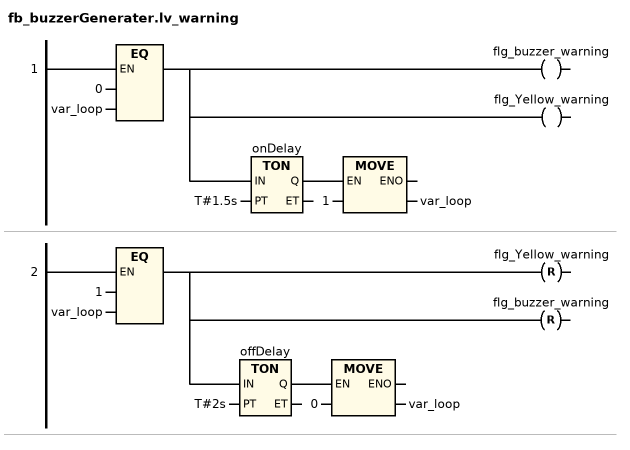
// NETWORK 1
_w3 := 0 = var_loop;
flg_buzzer_warning := _w3;
flg_Yellow_warning := _w3;
onDelay(IN := _w3, PT := T#1.5s); // TON
IF onDelay.Q THEN var_loop := 1; END_IF

// NETWORK 2
_w4 := 1 = var_loop;
flg_Yellow_warning R= _w4;
flg_buzzer_warning R= _w4;
offDelay(IN := _w4, PT := T#2s); // TON
IF offDelay.Q THEN var_loop := 0; END_IF
END_ACTION

ACTION manual:
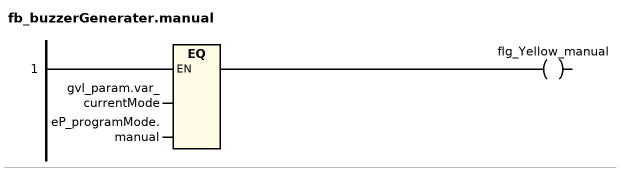
// NETWORK 1
flg_Yellow_manual := gvl_param.var_currentMode = eP_programMode.manual;
END_ACTION

END_FUNCTION_BLOCK

// ---- FBs/fb_eleControllers.TcPOU
FUNCTION_BLOCK fb_eleControllers
VAR_INPUT
END_VAR
VAR_OUTPUT
END_VAR
VAR
END_VAR

gvl_elecylinder.fbi_axisTransport(
	var_ref_ele:= gvl_elecylinder.ref_axis_transport, 
	in_flg_run:= , 
	in_var_moveMode:= , 
	in_flg_pause:= , 
	out_flg_run=> , 
	out_flg_busy=> , 
	out_flg_Done=> , 
	out_flg_error=> );
gvl_elecylinder.fbi_axisSample(
	var_ref_ele:= gvl_elecylinder.ref_axis_sample, 
	in_flg_run:= , 
	in_var_moveMode:= , 
	in_flg_pause:= NOT gvl_io.flg_frontSaftyDoor AND gvl_param.var_currentMode = eP_programMode.auto, 
	out_flg_run=> , 
	out_flg_busy=> , 
	out_flg_Done=> , 
	out_flg_error=> );
gvl_elecylinder.fbi_axisTrayChange(
	var_ref_ele:= gvl_elecylinder.ref_axis_trayChange, 
	in_flg_run:= , 
	in_var_moveMode:= , 
	in_flg_pause:=  NOT gvl_io.flg_frontSaftyDoor AND gvl_param.var_currentMode = eP_programMode.auto, 
	out_flg_run=> , 
	out_flg_busy=> , 
	out_flg_Done=> , 
	out_flg_error=> );
gvl_elecylinder.fbi_axisRotary(
	var_ref_ele:= gvl_elecylinder.ref_axis_rotary, 
	in_flg_run:= , 
	in_var_moveMode:= , 
	in_flg_pause:= , 
	out_flg_run=> , 
	out_flg_busy=> , 
	out_flg_Done=> , 
	out_flg_error=> );
gvl_elecylinder.fbi_gm_axisPickUp(
	var_ref_ele:= gvl_elecylinder.ref_gm_axisPickUp, 
	in_flg_run:= , 
	in_var_moveMode:= , 
	in_flg_pause:= , 
	out_flg_run=> , 
	out_flg_busy=> , 
	out_flg_Done=> , 
	out_flg_error=> );
gvl_elecylinder.fbi_gm_axisTransport(
	var_ref_ele:= gvl_elecylinder.ref_gm_axisTransport, 
	in_flg_run:= , 
	in_var_moveMode:= , 
	in_flg_pause:= , 
	out_flg_run=> , 
	out_flg_busy=> , 
	out_flg_Done=> , 
	out_flg_error=> );
	
IF gvl_elecylinder.ref_axis_trayChange.input.in_flg_sensA THEN
	gvl_param.var_currentTrayPos := 1;
	gvl_visu.var_currentTableMsg := "上段";
ELSIF gvl_elecylinder.ref_axis_trayChange.input.in_flg_sensB THEN
	gvl_param.var_currentTrayPos := 2;
	gvl_visu.var_currentTableMsg := "下段";
ELSE 
	gvl_param.var_currentTrayPos := 0;
	gvl_visu.var_currentTableMsg := "テーブル移動中...";
END_IF

END_FUNCTION_BLOCK

// ---- FBs/fb_svControllers.TcPOU
FUNCTION_BLOCK fb_svControllers
VAR_INPUT
END_VAR
VAR_OUTPUT
END_VAR
VAR
END_VAR

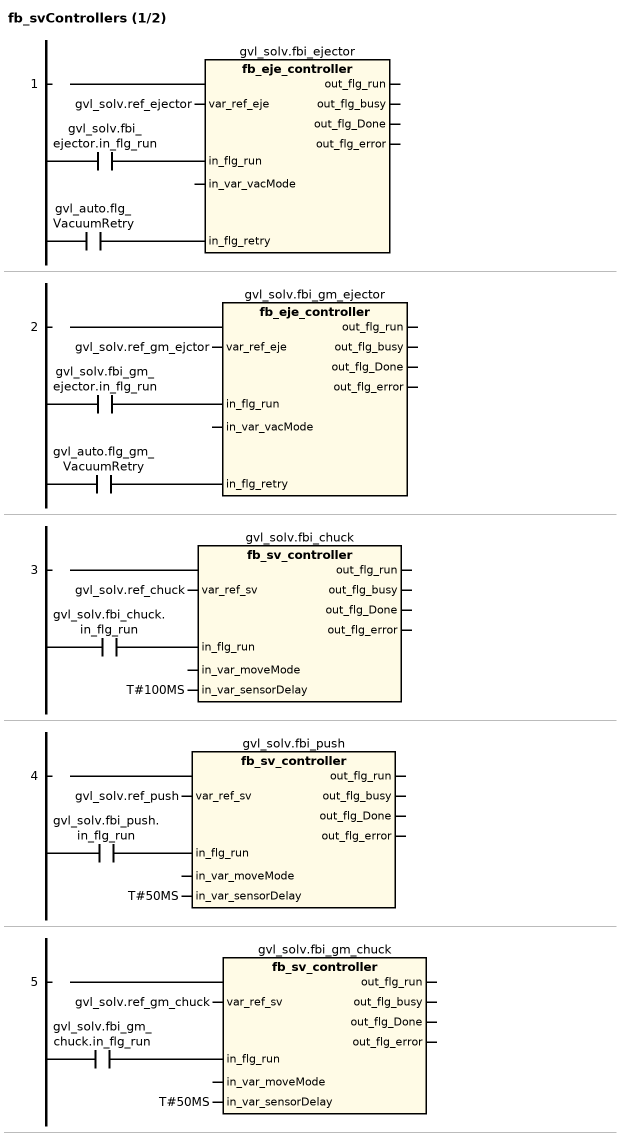
// NETWORK 1
gvl_solv.fbi_ejector(
    var_ref_eje := gvl_solv.ref_ejector,
    in_flg_run := gvl_solv.fbi_ejector.in_flg_run,
    in_flg_retry := gvl_auto.flg_VacuumRetry); // fb_eje_controller

// NETWORK 2
gvl_solv.fbi_gm_ejector(
    var_ref_eje := gvl_solv.ref_gm_ejctor,
    in_flg_run := gvl_solv.fbi_gm_ejector.in_flg_run,
    in_flg_retry := gvl_auto.flg_gm_VacuumRetry); // fb_eje_controller

// NETWORK 3
gvl_solv.fbi_chuck(
    var_ref_sv := gvl_solv.ref_chuck,
    in_flg_run := gvl_solv.fbi_chuck.in_flg_run,
    in_var_sensorDelay := T#100MS); // fb_sv_controller

// NETWORK 4
gvl_solv.fbi_push(
    var_ref_sv := gvl_solv.ref_push,
    in_flg_run := gvl_solv.fbi_push.in_flg_run,
    in_var_sensorDelay := T#50MS); // fb_sv_controller

// NETWORK 5
gvl_solv.fbi_gm_chuck(
    var_ref_sv := gvl_solv.ref_gm_chuck,
    in_flg_run := gvl_solv.fbi_gm_chuck.in_flg_run,
    in_var_sensorDelay := T#50MS); // fb_sv_controller

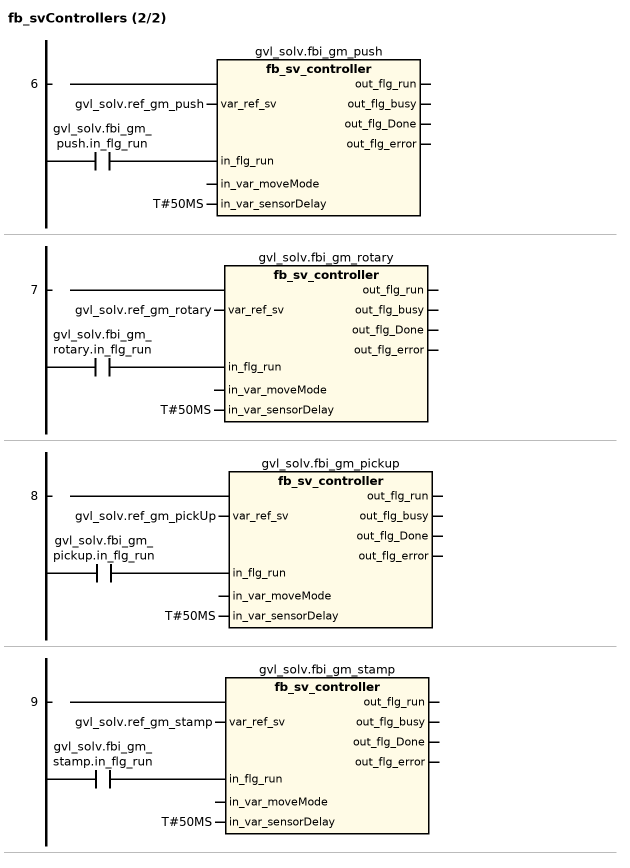
// NETWORK 6
gvl_solv.fbi_gm_push(
    var_ref_sv := gvl_solv.ref_gm_push,
    in_flg_run := gvl_solv.fbi_gm_push.in_flg_run,
    in_var_sensorDelay := T#50MS); // fb_sv_controller

// NETWORK 7
gvl_solv.fbi_gm_rotary(
    var_ref_sv := gvl_solv.ref_gm_rotary,
    in_flg_run := gvl_solv.fbi_gm_rotary.in_flg_run,
    in_var_sensorDelay := T#50MS); // fb_sv_controller

// NETWORK 8
gvl_solv.fbi_gm_pickup(
    var_ref_sv := gvl_solv.ref_gm_pickUp,
    in_flg_run := gvl_solv.fbi_gm_pickup.in_flg_run,
    in_var_sensorDelay := T#50MS); // fb_sv_controller

// NETWORK 9
gvl_solv.fbi_gm_stamp(
    var_ref_sv := gvl_solv.ref_gm_stamp,
    in_flg_run := gvl_solv.fbi_gm_stamp.in_flg_run,
    in_var_sensorDelay := T#50MS); // fb_sv_controller

END_FUNCTION_BLOCK

// ---- FBs/fb_ejecter/fb_eje_controller.TcPOU
FUNCTION_BLOCK fb_eje_controller
VAR_IN_OUT
	var_ref_eje : ref_eje_io;
END_VAR
VAR_INPUT
	in_flg_run : BOOL;
	in_var_vacMode : eP_ejeVacMode;
	in_flg_retry: BOOL;
END_VAR
VAR_OUTPUT
	out_flg_run : BOOL;
	out_flg_busy: BOOL;
	out_flg_Done: BOOL;
	out_flg_error : BOOL;
END_VAR
VAR
	var_buf_moveMode: eP_ejeVacMode;
	flg_vacOnDone: BOOL;
	flg_vacOffDone: BOOL;
	flg_vacBreakDone: BOOL;
	flg_vacHaltDone: BOOL;
	fbi_brakTime: TON;
	flg_breakDone: BOOL;
	var_timeOut: TON;
	in: BOOL;
END_VAR
VAR // added by the converter: edge detectors and wires of the graphical bodies
    _rt1, _rt2, _rt3, _rt4 : R_TRIG;
    _w1, _w2, _w3, _w4, _w5 : BOOL;
END_VAR

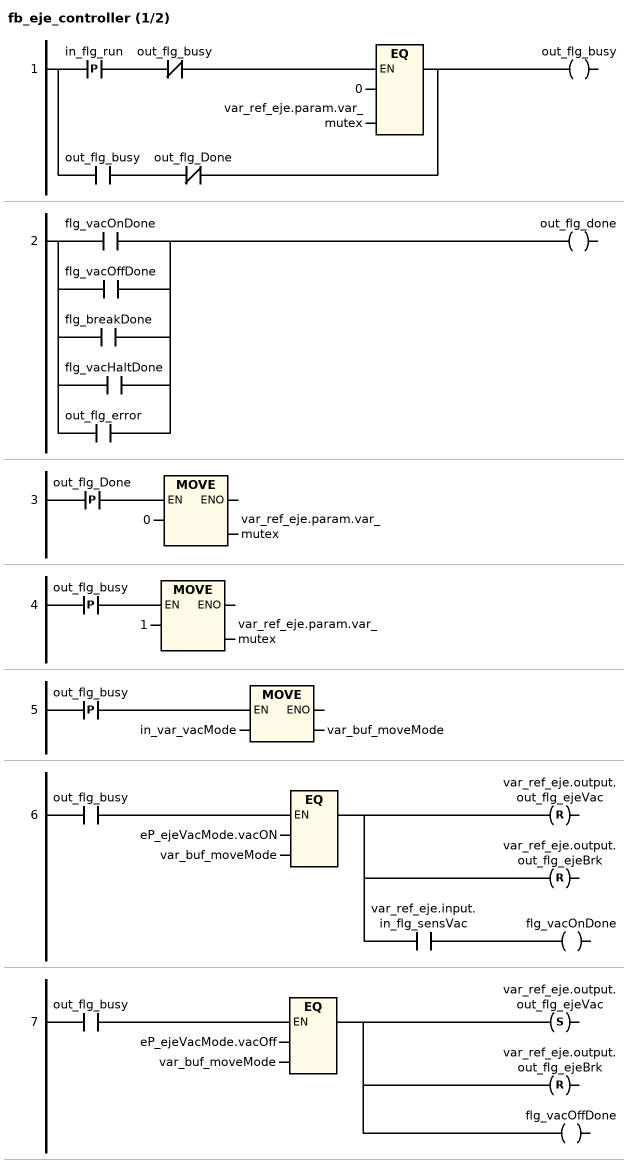
// NETWORK 1
_rt1(CLK := in_flg_run);
out_flg_busy := _rt1.Q AND NOT out_flg_busy AND 0 = var_ref_eje.param.var_mutex OR out_flg_busy AND NOT out_flg_Done;

// NETWORK 2
out_flg_done := flg_vacOnDone OR flg_vacOffDone OR flg_breakDone OR flg_vacHaltDone OR out_flg_error;

// NETWORK 3
_rt2(CLK := out_flg_Done);
IF _rt2.Q THEN var_ref_eje.param.var_mutex := 0; END_IF

// NETWORK 4
_rt3(CLK := out_flg_busy);
IF _rt3.Q THEN var_ref_eje.param.var_mutex := 1; END_IF

// NETWORK 5
_rt4(CLK := out_flg_busy);
IF _rt4.Q THEN var_buf_moveMode := in_var_vacMode; END_IF

// NETWORK 6
_w1 := out_flg_busy AND eP_ejeVacMode.vacON = var_buf_moveMode;
var_ref_eje.output.out_flg_ejeVac R= _w1;
var_ref_eje.output.out_flg_ejeBrk R= _w1;
flg_vacOnDone := _w1 AND var_ref_eje.input.in_flg_sensVac;

// NETWORK 7
_w2 := out_flg_busy AND eP_ejeVacMode.vacOff = var_buf_moveMode;
var_ref_eje.output.out_flg_ejeVac S= _w2;
var_ref_eje.output.out_flg_ejeBrk R= _w2;
flg_vacOffDone := _w2;

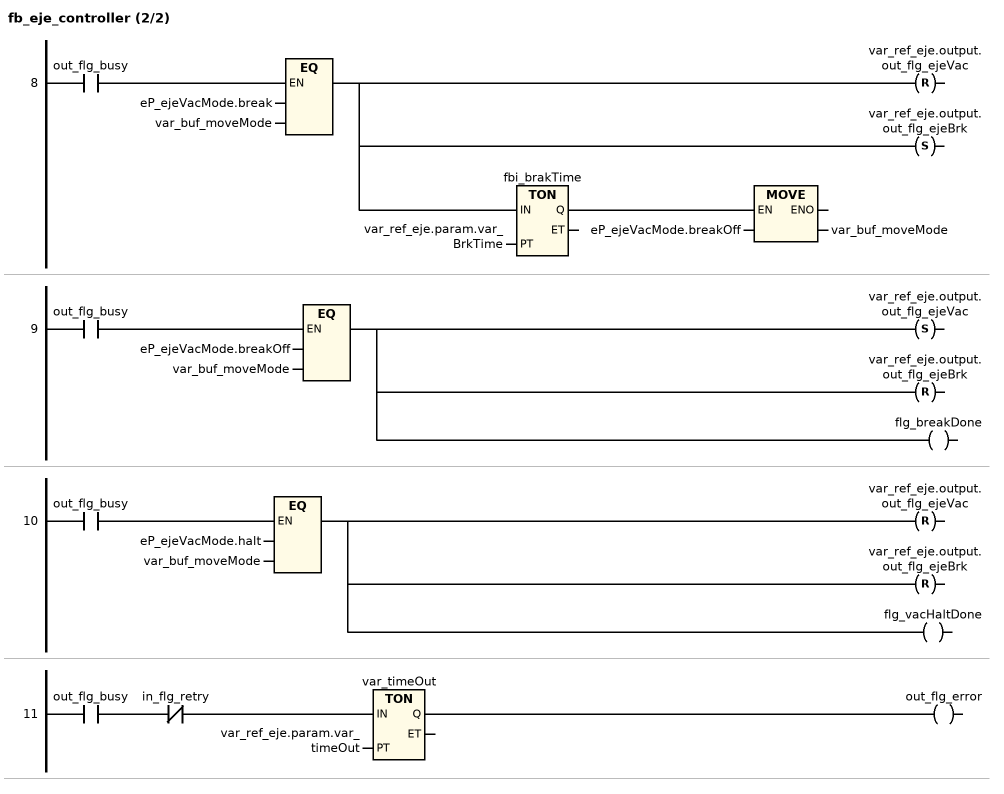
// NETWORK 8
_w3 := out_flg_busy AND eP_ejeVacMode.break = var_buf_moveMode;
var_ref_eje.output.out_flg_ejeVac R= _w3;
var_ref_eje.output.out_flg_ejeBrk S= _w3;
fbi_brakTime(IN := _w3, PT := var_ref_eje.param.var_BrkTime); // TON
IF fbi_brakTime.Q THEN var_buf_moveMode := eP_ejeVacMode.breakOff; END_IF

// NETWORK 9
_w4 := out_flg_busy AND eP_ejeVacMode.breakOff = var_buf_moveMode;
var_ref_eje.output.out_flg_ejeVac S= _w4;
var_ref_eje.output.out_flg_ejeBrk R= _w4;
flg_breakDone := _w4;

// NETWORK 10
_w5 := out_flg_busy AND eP_ejeVacMode.halt = var_buf_moveMode;
var_ref_eje.output.out_flg_ejeVac R= _w5;
var_ref_eje.output.out_flg_ejeBrk R= _w5;
flg_vacHaltDone := _w5;

// NETWORK 11
var_timeOut(IN := out_flg_busy AND NOT in_flg_retry, PT := var_ref_eje.param.var_timeOut); // TON
out_flg_error := var_timeOut.Q;

END_FUNCTION_BLOCK

// ---- FBs/fb_sv/fb_sv_controller.TcPOU
FUNCTION_BLOCK fb_sv_controller
VAR_IN_OUT
	var_ref_sv : ref_sv_io;
END_VAR
VAR_INPUT
	in_flg_run : BOOL;
	in_var_moveMode : eP_svMoveMode;
	in_var_sensorDelay : TIME;
END_VAR
VAR_OUTPUT
	out_flg_run : BOOL;
	out_flg_busy: BOOL;
	out_flg_Done: BOOL;
	out_flg_error : BOOL;
END_VAR
VAR
	var_buf_moveMode: eP_svMoveMode;
	fbi_sensorDelayTimerA: TON;
	fbi_sensorDelayTimerB: TON;
	flg_svADone: BOOL;
	flg_svBDone: BOOL;
	fbi_timeOut: TON;
	flg_svSDone: BOOL;
END_VAR
VAR // added by the converter: edge detectors and wires of the graphical bodies
    _rt1, _rt2, _rt3, _rt4 : R_TRIG;
    _w1, _w2, _w3 : BOOL;
END_VAR

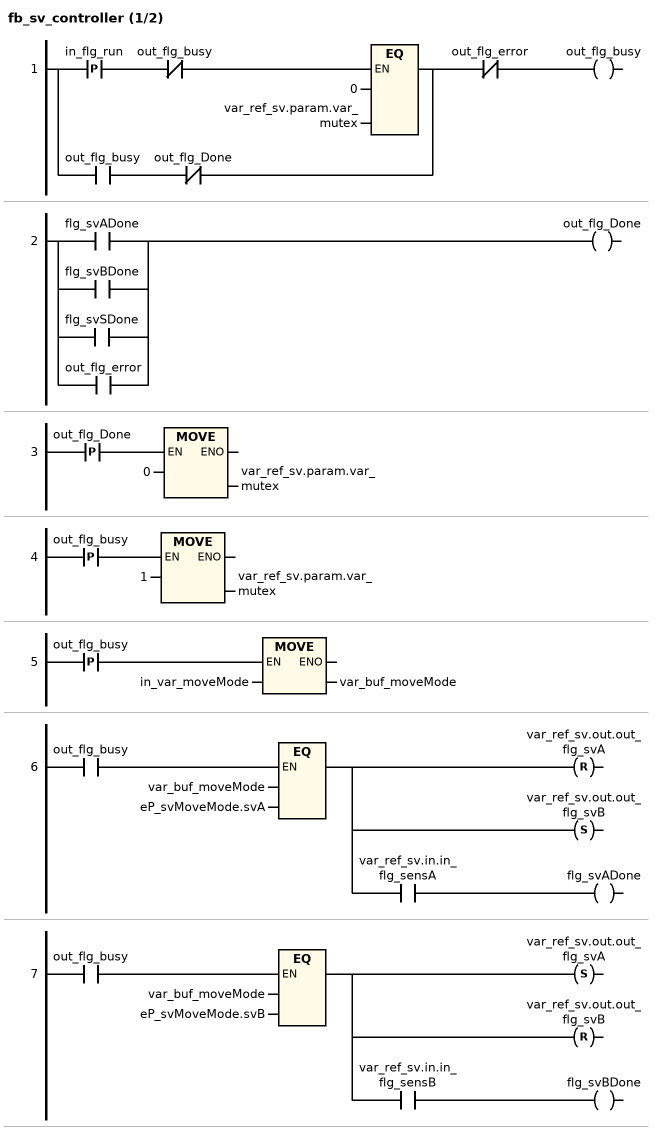
// NETWORK 1
_rt1(CLK := in_flg_run);
out_flg_busy := (_rt1.Q AND NOT out_flg_busy AND 0 = var_ref_sv.param.var_mutex OR out_flg_busy AND NOT out_flg_Done) AND NOT out_flg_error;

// NETWORK 2
out_flg_Done := flg_svADone OR flg_svBDone OR flg_svSDone OR out_flg_error;

// NETWORK 3
_rt2(CLK := out_flg_Done);
IF _rt2.Q THEN var_ref_sv.param.var_mutex := 0; END_IF

// NETWORK 4
_rt3(CLK := out_flg_busy);
IF _rt3.Q THEN var_ref_sv.param.var_mutex := 1; END_IF

// NETWORK 5
_rt4(CLK := out_flg_busy);
IF _rt4.Q THEN var_buf_moveMode := in_var_moveMode; END_IF

// NETWORK 6
_w1 := out_flg_busy AND var_buf_moveMode = eP_svMoveMode.svA;
var_ref_sv.out.out_flg_svA R= _w1;
var_ref_sv.out.out_flg_svB S= _w1;
flg_svADone := _w1 AND var_ref_sv.in.in_flg_sensA;

// NETWORK 7
_w2 := out_flg_busy AND var_buf_moveMode = eP_svMoveMode.svB;
var_ref_sv.out.out_flg_svA S= _w2;
var_ref_sv.out.out_flg_svB R= _w2;
flg_svBDone := _w2 AND var_ref_sv.in.in_flg_sensB;

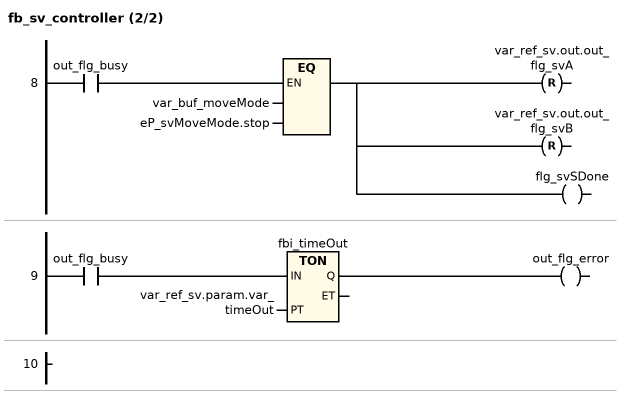
// NETWORK 8
_w3 := out_flg_busy AND var_buf_moveMode = eP_svMoveMode.stop;
var_ref_sv.out.out_flg_svA R= _w3;
var_ref_sv.out.out_flg_svB R= _w3;
flg_svSDone := _w3;

// NETWORK 9
fbi_timeOut(IN := out_flg_busy, PT := var_ref_sv.param.var_timeOut); // TON
out_flg_error := fbi_timeOut.Q;

// NETWORK 10

END_FUNCTION_BLOCK

// ---- FBs/fb_sampleSchedule.TcPOU
FUNCTION_BLOCK fb_sampleSchedule
VAR_INPUT
	in_var_enableSchedule: ARRAY[0..6] OF BOOL;
	in_var_scheduleTimeH : ARRAY[0..6] OF WORD;
	in_var_scheduleTimeM : ARRAY[0..6] OF WORD;
END_VAR
VAR_OUTPUT
	out_flg_sampletriger : bool;
END_VAR
VAR
	fbi_GetLocalAmsNetId : FB_GetLocalAmsNetId;
	fbi_LocalSystemTime : FB_LocalSystemTime;
	var_scheduleTime : ARRAY[0..6] OF s_timeSchedule;
	var_scheduleNumber : INT;
	fbi_r_trig: R_TRIG;
	var_process: INT;
END_VAR

fbi_GetLocalAmsNetId(
	bExecute:= TRUE, 
	tTimeOut:= , 
	bBusy=> , 
	bError=> , 
	nErrId=> , 
	AddrString=> , 
	AddrBytes=> );
fbi_LocalSystemTime(
	sNetID:=fbi_GetLocalAmsNetId.AddrString , 
	bEnable:= TRUE, 
	dwCycle:= , 
	dwOpt:= , 
	tTimeout:= , 
	bValid=> , 
	systemTime=> ,
	tzID=> );
fbi_r_trig(CLK:= , Q=> );
FOR var_scheduleNumber := 0 TO 6 BY 1 DO
	IF in_var_enableSchedule[var_scheduleNumber] THEN
		var_scheduleTime[var_scheduleNumber].hour := in_var_scheduleTimeH[var_scheduleNumber];
		var_scheduleTime[var_scheduleNumber].minute := in_var_scheduleTimeM[var_scheduleNumber];
		IF fbi_LocalSystemTime.systemTime.wHour = var_scheduleTime[var_scheduleNumber].hour THEN
			IF fbi_LocalSystemTime.systemTime.wMinute = var_scheduleTime[var_scheduleNumber].minute THEN		
				fbi_r_trig.CLK := TRUE;
			ELSE
				fbi_r_trig.CLK := FALSE;
			END_IF
		END_IF
	END_IF
END_FOR
out_flg_sampletriger := fbi_r_trig.Q;

END_FUNCTION_BLOCK

// ---- FBs/fb_text_control.TcPOU
FUNCTION_BLOCK fb_text_control
VAR_INPUT
END_VAR
VAR_OUTPUT
END_VAR
VAR
END_VAR

IF gvl_param.var_currentMode = eP_programMode.auto THEN
	IF gvl_debug.out_busy THEN
		gvl_text.var_auto_runing := "デバッグ運転中";
	ELSE
		gvl_text.var_auto_runing := "自動運転中";
	END_IF
ELSE
	gvl_text.var_auto_runing := "自動運転開始";
END_IF
IF gvl_auto.autoModeStop THEN
	gvl_text.var_stopping:= "自動運転停止中";
ELSE
	gvl_text.var_stopping:= "自動運転停止";
END_IF
IF gvl_visu.flg_btn_trayChangeDone THEN
	gvl_text.var_trayChangeDone:= "トレイ交換完了済";
ELSE
	gvl_text.var_trayChangeDone:= "トレイ交換完了";
END_IF

END_FUNCTION_BLOCK

// ---- FBs/fb_motionController.TcPOU
FUNCTION_BLOCK fb_motionController
VAR_INPUT
	in_flg_run : BOOL;
END_VAR
VAR_OUTPUT
	out_flg_run : BOOL;
END_VAR
VAR_IN_OUT
	var_ref_X : ref_mc_moveAbs;
	var_ref_Y : ref_mc_moveAbs;
	var_ref_Z : ref_mc_moveAbs;
END_VAR
VAR_INPUT
	in_flg_start : BOOL;
	in_var_targetPosX : LREAL;
	in_var_targetPosY : LREAL;
	in_var_targetPosZ : LREAL;
	in_var_direction : eP_motionDirection;
	
END_VAR
VAR_OUTPUT
	out_flg_busy : BOOL;
	out_flg_Done : BOOL;
	out_flg_moveXYDone : BOOL;
	
END_VAR
VAR
	SFCInit : BOOL;
	fbi_r_TIRG: R_TRIG;
	fbi_f_TRIG: F_TRIG;
	var_buf_targetPosX: LREAL;
	var_buf_targetPosY: LREAL;
	var_buf_targetPosZ: LREAL;
	var_buf_direction: eP_motionDirection;
	trn_getParamDone: BOOL;
	var_mutex: INT;
	trn_moveXY_1Done: BOOL;
	trn_moveZ_1Done: BOOL;
	trn_moveZ_2Done: BOOL;
	trn_moveXY_2Done: BOOL;
	
	trn_moveX_3Done: BOOL;
	trn_moveY_3Done: BOOL;
	trn_moveZ_3Done: BOOL;
	
	trn_moveX_4Done: BOOL;
	trn_moveY_4Done: BOOL;
	trn_moveZ_4Done: BOOL;

	trn_executeReset2Done: BOOL;
	var_process: INT;
END_VAR

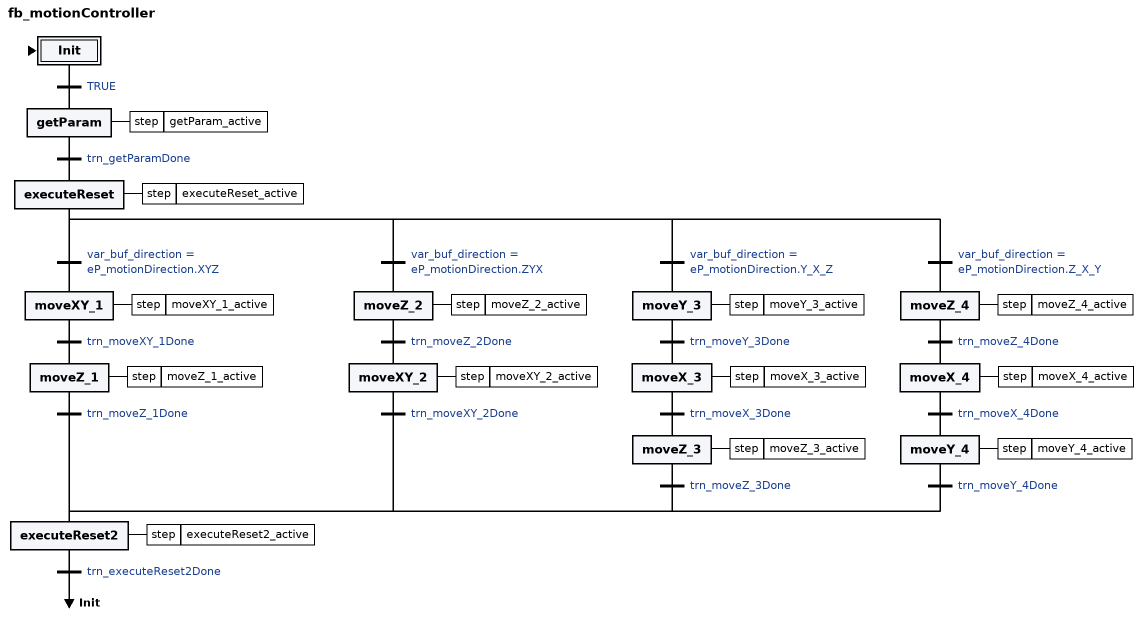
INITIAL_STEP Init:
END_STEP
TRANSITION FROM Init TO getParam
    := TRUE;
END_TRANSITION
STEP getParam:
    getParam_active(N);  // step action
END_STEP
TRANSITION FROM getParam TO executeReset
    := trn_getParamDone;
END_TRANSITION
STEP executeReset:
    executeReset_active(N);  // step action
END_STEP
TRANSITION FROM executeReset TO moveXY_1
    := var_buf_direction = eP_motionDirection.XYZ;
END_TRANSITION
STEP moveXY_1:
    moveXY_1_active(N);  // step action
END_STEP
TRANSITION FROM moveXY_1 TO moveZ_1
    := trn_moveXY_1Done;
END_TRANSITION
STEP moveZ_1:
    moveZ_1_active(N);  // step action
END_STEP
TRANSITION FROM moveZ_1 TO executeReset2
    := trn_moveZ_1Done;
END_TRANSITION
TRANSITION FROM executeReset TO moveZ_2
    := var_buf_direction = eP_motionDirection.ZYX;
END_TRANSITION
STEP moveZ_2:
    moveZ_2_active(N);  // step action
END_STEP
TRANSITION FROM moveZ_2 TO moveXY_2
    := trn_moveZ_2Done;
END_TRANSITION
STEP moveXY_2:
    moveXY_2_active(N);  // step action
END_STEP
TRANSITION FROM moveXY_2 TO executeReset2
    := trn_moveXY_2Done;
END_TRANSITION
TRANSITION FROM executeReset TO moveY_3
    := var_buf_direction = eP_motionDirection.Y_X_Z;
END_TRANSITION
STEP moveY_3:
    moveY_3_active(N);  // step action
END_STEP
TRANSITION FROM moveY_3 TO moveX_3
    := trn_moveY_3Done;
END_TRANSITION
STEP moveX_3:
    moveX_3_active(N);  // step action
END_STEP
TRANSITION FROM moveX_3 TO moveZ_3
    := trn_moveX_3Done;
END_TRANSITION
STEP moveZ_3:
    moveZ_3_active(N);  // step action
END_STEP
TRANSITION FROM moveZ_3 TO executeReset2
    := trn_moveZ_3Done;
END_TRANSITION
TRANSITION FROM executeReset TO moveZ_4
    := var_buf_direction = eP_motionDirection.Z_X_Y;
END_TRANSITION
STEP moveZ_4:
    moveZ_4_active(N);  // step action
END_STEP
TRANSITION FROM moveZ_4 TO moveX_4
    := trn_moveZ_4Done;
END_TRANSITION
STEP moveX_4:
    moveX_4_active(N);  // step action
END_STEP
TRANSITION FROM moveX_4 TO moveY_4
    := trn_moveX_4Done;
END_TRANSITION
STEP moveY_4:
    moveY_4_active(N);  // step action
END_STEP
TRANSITION FROM moveY_4 TO executeReset2
    := trn_moveY_4Done;
END_TRANSITION
STEP executeReset2:
    executeReset2_active(N);  // step action
END_STEP
TRANSITION FROM executeReset2 TO Init
    := trn_executeReset2Done;
END_TRANSITION

ACTION executeReset_active:
IF executeReset._x AND executeReset.x = FALSE THEN
	var_ref_x.Execute := FALSE;
	var_ref_y.Execute := FALSE;
	var_ref_z.Execute := FALSE;
ELSIF executeReset._x AND executeReset.x THEN
	var_ref_x.Execute := FALSE;
	var_ref_y.Execute := FALSE;
	var_ref_z.Execute := FALSE;
END_IF
END_ACTION

ACTION executeReset2_active:
IF executeReset2._x AND executeReset2.x= FALSE THEN
	trn_executeReset2Done := FALSE;
	var_ref_x.Execute := FALSE;
	var_ref_y.Execute := FALSE;
	var_ref_z.Execute := FALSE;
	out_flg_done := TRUE;
	out_flg_moveXYDone := FALSE;
ELSIF executeReset2._x AND executeReset2.x THEN
	var_ref_x.Execute := FALSE;
	var_ref_y.Execute := FALSE;
	var_ref_z.Execute := FALSE;
	trn_executeReset2Done := TRUE;
	out_flg_done := FALSE;
	in_flg_start := FALSE;
END_IF
END_ACTION

ACTION getParam_active:
fbi_r_TIRG(CLK:= in_flg_start, Q=> );
IF getParam._x AND getParam.x = FALSE THEN
	var_mutex := 0;
	trn_getParamDone := FALSE;
	out_flg_moveXYDone:= FALSE;
	in_flg_start := FALSE;
ELSIF getParam._x AND getParam.x THEN
	IF fbi_r_TIRG.Q THEN
		var_ref_x.Position := in_var_targetPosX;
		var_ref_Y.Position := in_var_targetPosY;
		var_ref_Z.Position := in_var_targetPosZ;
		var_buf_direction := in_var_direction;
		var_mutex := 1;
	END_IF
	IF var_mutex = 1 THEN
		out_flg_busy := TRUE;
		trn_getParamDone := TRUE;
	ELSE
		out_flg_busy := FALSE;
		trn_getParamDone := FALSE;
	END_IF
	IF in_flg_run THEN
		out_flg_run := TRUE;
	ELSE
		out_flg_run := FALSE;
	END_IF
END_IF
END_ACTION

ACTION moveX_3_active:
IF moveX_3._x AND moveX_3.x = FALSE THEN
	trn_moveX_3Done := FALSE;
	var_process := 0;
ELSIF moveX_3._x AND moveX_3.x THEN
	CASE var_process OF
		0:
			var_ref_x.Execute := TRUE;
			var_process := 1;
		1:
			IF var_ref_x.Done THEN
				trn_moveX_3Done := TRUE;
			END_IF
	END_CASE
END_IF
END_ACTION

ACTION moveX_4_active:
IF moveX_4._x AND moveX_4.x = FALSE THEN
	trn_moveX_4Done := FALSE;
	var_process := 0;
ELSIF moveX_4._x AND moveX_4.x THEN
	CASE var_process OF
		0:
			var_ref_x.Execute := TRUE;
			var_process := 1;
		1:
			IF var_ref_x.Done THEN
				trn_moveX_4Done := TRUE;
			END_IF
	END_CASE
END_IF
END_ACTION

ACTION moveXY_1_active:
IF moveXY_1._x AND moveXY_1.x = FALSE THEN
	out_flg_moveXYDone:= FALSE;
	trn_moveXY_1Done := FALSE;
	var_process := 0;
ELSIF moveXY_1._x AND moveXY_1.x THEN
	CASE var_process OF
		0:
			var_ref_x.Execute := TRUE;
			var_ref_y.Execute := TRUE;
			var_process := 1;
		1:
			IF var_ref_x.Done AND var_ref_y.Done THEN
				out_flg_moveXYDone:= TRUE;
				trn_moveXY_1Done := TRUE;
			END_IF
	END_CASE
END_IF
END_ACTION

ACTION moveXY_2_active:
IF moveXY_2._x AND moveXY_2.x = FALSE THEN
	trn_moveXY_2Done := FALSE;
	var_process := 0;
ELSIF moveXY_2._x AND moveXY_2.x THEN
	CASE var_process OF
		0:
			var_ref_x.Execute := TRUE;
			var_ref_y.Execute := TRUE;
			var_process := 1;
		1:
			IF var_ref_x.Done AND var_ref_y.Done THEN
				trn_moveXY_2Done := TRUE;
			END_IF
	END_CASE
END_IF
END_ACTION

ACTION moveY_3_active:
IF moveY_3._x AND moveY_3.x = FALSE THEN
	trn_moveY_3Done := FALSE;
	var_process := 0;
ELSIF moveY_3._x AND moveY_3.x THEN
	CASE var_process OF
		0:
			var_ref_y.Execute := TRUE;
			var_process := 1;
		1:
			IF var_ref_y.Done THEN
				trn_moveY_3Done := TRUE;
			END_IF
	END_CASE
END_IF
END_ACTION

ACTION moveY_4_active:
IF moveY_4._x AND moveY_4.x = FALSE THEN
	trn_moveY_4Done := FALSE;
	var_process := 0;
ELSIF moveY_4._x AND moveY_4.x THEN
	CASE var_process OF
		0:
			var_ref_y.Execute := TRUE;
			var_process := 1;
		1:
			IF var_ref_y.Done THEN
				trn_moveY_4Done := TRUE;
			END_IF
	END_CASE
END_IF
END_ACTION

ACTION moveZ_1_active:
IF moveZ_1._x AND moveZ_1.x = FALSE THEN
	out_flg_moveXYDone := FALSE;
	trn_moveZ_1Done := FALSE;
	var_process := 0;
ELSIF moveZ_1._x AND moveZ_1.x THEN
	CASE var_process OF
		0:
			var_ref_z.Execute := TRUE;
			var_process := 1;
		1:
			IF var_ref_z.Done THEN
				trn_moveZ_1Done := TRUE;
			END_IF
	END_CASE
	

END_IF
END_ACTION

ACTION moveZ_2_active:
IF moveZ_2._x AND moveZ_2.x = FALSE THEN
	trn_moveZ_2Done := FALSE;
	var_process := 0;
ELSIF moveZ_2._x AND moveZ_2.x THEN
	CASE var_process OF
		0:
			var_ref_z.Execute := TRUE;
			var_process := 1;
		1:
			IF var_ref_z.Done THEN
				trn_moveZ_2Done := TRUE;
			END_IF
	END_CASE
END_IF
END_ACTION

ACTION moveZ_3_active:
IF moveZ_3._x AND moveZ_3.x = FALSE THEN
	trn_moveZ_3Done := FALSE;
	var_process := 0;
ELSIF moveZ_3._x AND moveZ_3.x THEN
	CASE var_process OF
		0:
			var_ref_Z.Execute := TRUE;
			var_process := 1;
		1:
			IF var_ref_Z.Done THEN
				trn_moveZ_3Done := TRUE;
			END_IF
	END_CASE
END_IF
END_ACTION

ACTION moveZ_4_active:
IF moveZ_4._x AND moveZ_4.x = FALSE THEN
	trn_moveZ_4Done := FALSE;
	var_process := 0;
ELSIF moveZ_4._x AND moveZ_4.x THEN
	CASE var_process OF
		0:
			var_ref_z.Execute := TRUE;
			var_process := 1;
		1:
			IF var_ref_z.Done THEN
				trn_moveZ_4Done := TRUE;
			END_IF
	END_CASE
END_IF
END_ACTION

PROPERTY p_Init : bool
GET
p_init := THIS^.SFCInit;
END_GET
SET
THIS^.SFCInit := p_init;
END_SET
END_PROPERTY

END_FUNCTION_BLOCK

// ---- FBs/error/fun_setAlarm.TcPOU
FUNCTION fun_setAlarm : bool
VAR_INPUT
	in_flg_set : BOOL;
	in_flg_reset : BOOL;
END_VAR
VAR

END_VAR


	IF in_flg_reset = FALSE THEN
		IF in_flg_set THEN
			fun_setAlarm := TRUE;
		END_IF
	ELSIF in_flg_reset THEN
		fun_setAlarm := FALSE;
	END_IF

END_FUNCTION

// ---- GlobalTextList.TcGTLO
TEXTLIST GlobalTextList
  137 = '\tメイン'
  1405 = '   メッセージ:  %s '
  105 = ' %1.2f'
  57 = '# %u'
  85 = '#1: %d'
  201 = '#2: %d'
  1664 = '#3: %d'
  935 = '#4: %d'
  388 = '#5: %d'
  1230 = '#6: %d'
  1322 = '#7: %d'
  1159 = '#8: %d'
  1616 = '%10'
  997 = '%10.2f'
  736 = '%10.2f  °'
  813 = '%10.2f mm'
  14 = '%2'
  1332 = '%2d'
  315 = '%3.2f mm'
  142 = '%4.2f mm'
  300 = '%d'
  714 = '%d '
  745 = '%s'
  810 = '+'
  462 = '-'
  2287 = '/'
  756 = '4         3         2         1'
  944 = '<'
  1456 = '>'
  622 = 'Back'
  814 = 'Cancel'
  472 = 'Cav1'
  1274 = 'Cav2'
  1277 = 'Cav3'
  682 = 'Cav4'
  1835 = 'Cav5'
  1513 = 'Cav6'
  1387 = 'Cav7'
  322 = 'Cav8'
  663 = 'CCW↺'
  457 = 'CLR'
  34 = 'CW↻'
  553 = 'Deactivate Robot'
  1196 = 'Deactivate sensor'
  1400 = 'debug'
  1321 = 'Debuger execute'
  1335 = 'Error'
  1392 = 'g'
  1204 = 'Gate OK'
  1401 = 'gvl_error.var_ary_alarmlistLog[INDEX].var_alarmLevel'
  1199 = 'incjet deney'
  352 = 'incjet deny'
  170 = 'incjet Done'
  531 = 'incjet ready'
  724 = 'incjetvDone'
  1136 = 'No'
  273 = 'O'
  96 = 'P'
  1025 = 'Palletize additonal mode'
  467 = 'Q'
  1112 = 'reset project'
  1066 = 'Run'
  1339 = 'Start'
  99 = 't'
  718 = 'X'
  314 = 'X軸'
  777 = 'x軸'
  319 = 'Y'
  511 = 'Yes'
  225 = 'Y軸'
  666 = 'y軸'
  160 = 'Z'
  788 = 'Z軸'
  858 = 'z軸'
  886 = 'θ軸'
  760 = '※手動運転時のみ'
  410 = '「ストッカ」\u3000チャック動作手順\u30000:チャック→押す→チャック\u3000/\u30001:押す→チャック→押す'
  326 = '「ストッカ」チャック動作手順'
  623 = '「ストッカ」チャック動作手順\u30000:チャック→押す→チャック/1:押す→チャック→押す'
  1188 = '「ストッカ」チャック動作手順\u30000:チャック→押す→チャック\u3000/\u30001:押す→チャック→押す'
  440 = '「測定」\u3000チャック動作手順\u30000:チャック→押す→チャック\u3000/\u30001:押す→チャック→押す'
  2005 = '「測定」チャック動作手順\u30000:チャック→押す→チャック\u3000/\u30001:押す→チャック→押す'
  22 = 'アラーム'
  141 = 'アラームリセット'
  86 = 'アラーム名'
  1268 = 'インクジェットメッセージ番号'
  1734 = 'インクジェット原点'
  761 = 'インクジェット可動点'
  179 = 'インクジェット有り'
  1603 = 'インクジェット横軸原点'
  1422 = 'インクジェット横軸可動点'
  164 = 'インチ'
  389 = 'エラーID'
  1227 = 'エラーログ'
  9 = 'キャビ数'
  1878 = 'キャビ番号:# %d'
  570 = 'ゲート上限'
  217 = 'ゲート下限'
  586 = 'ゲート測定OK信号'
  806 = 'ゲート測定モジュール'
  229 = 'ゲート測定モジュール有り'
  369 = 'ゲート長さ上限'
  358 = 'ゲート長さ下限'
  489 = 'サンプルスケジュール'
  785 = 'サンプルスケジュール設定'
  1341 = 'サンプルティーチング'
  95 = 'サンプル取り開始'
  256 = 'サンプル受け取り軸'
  832 = 'サンプル台にレンズがないことを'
  924 = 'サンプル台にレンズがないことを確認してください。'
  162 = 'ジョグ'
  118 = 'ストッカまで'
  1426 = 'ストッカファイバーセンサー'
  1363 = 'ストッカー側ゲート測定無し'
  83 = 'セット位置'
  1171 = 'センサー無効'
  449 = 'ダミー信号'
  689 = 'チャック測定閉'
  114 = 'チャック測定開'
  1071 = 'チャック閉'
  947 = 'チャック開'
  251 = 'ティーチング'
  25 = 'ティーチングデータを保存します。'
  1732 = 'デバッグ'
  224 = 'デバッグ開始'
  1390 = 'データ'
  382 = 'トレイ交換完了'
  1307 = 'トレイ交換完了済'
  1043 = 'トレイ横数'
  328 = 'トレイ歯抜け有り'
  263 = 'トレイ縦数'
  401 = 'トレー交換軸'
  293 = 'パレタイズをリセットします。'
  738 = 'パレタイズリセット'
  307 = 'ピックアップ位置'
  1247 = 'ピックアップ軸原点'
  1131 = 'ピックアップ軸可動点'
  283 = 'ブザー無効'
  368 = 'ポケット番号'
  163 = 'ポケット移動'
  1329 = 'メイン'
  767 = 'モニター'
  19 = 'モーター電源'
  975 = 'レンズセット完了信号'
  743 = 'レンズ取り位置'
  252 = 'レンズ取り位置移動'
  2270 = 'レンズ取得済'
  381 = 'レンズ受け取り回転軸'
  452 = 'レンズ受け取り軸横'
  507 = 'レンズ抑え閉'
  620 = 'レンズ抑え開'
  1271 = 'レンズ測定閉'
  787 = 'レンズ測定開'
  616 = 'レンズ要求信号'
  456 = '不良数'
  1952 = '使用有無'
  455 = '保存'
  236 = '入り数'
  2014 = '全ポケット移動'
  2205 = '全ポケット移動中'
  1062 = '分'
  763 = '初期位置'
  849 = '初期位置移動'
  284 = '単位/mm'
  1650 = '単位/°'
  1639 = '単位10μ'
  1743 = '印字ユニット有り'
  139 = '原点'
  2198 = '受取完了'
  882 = '可動点'
  2084 = '各製品共通設定'
  325 = '吸着OFF'
  468 = '吸着ON'
  366 = '品種選択'
  232 = '品質確認'
  59 = '回転軸不使用'
  285 = '回転軸原点'
  166 = '回転軸原点逆転'
  350 = '回転軸可動点'
  316 = '回転軸自動運転動作不使用'
  1280 = '安全扉開放中'
  257 = '手動サンプル取り開始'
  339 = '手動速度X: %d mm/s'
  1841 = '手動速度Y: %d mm/s'
  1304 = '手動速度Z: %d mm/s'
  847 = '手動速度θ:[%d]度/s'
  1116 = '手動運転'
  857 = '捨て位置'
  910 = '捨て位置移動'
  662 = '搬送軸原点'
  582 = '搬送軸可動点'
  754 = '時'
  984 = '書き込み'
  451 = '横'
  715 = '測定まで'
  238 = '測定ファイバーセンサー'
  1601 = '現在値'
  367 = '現在値㎜'
  936 = '番号'
  1007 = '発生中エラー'
  200 = '発生時刻'
  82 = '登録番号'
  823 = '破壊'
  1417 = '確認してください。'
  172 = '移動'
  2196 = '移動中'
  850 = '移動停止'
  969 = '縦'
  165 = '自動加速度X: %d mm/s²'
  133 = '自動加速度Y: %d mm/s²'
  870 = '自動加速度Z: %d mm/s²'
  205 = '自動加速度θ:[%d]mm/s²'
  494 = '自動減速度X: %d mm/s²'
  643 = '自動減速度Y: %d mm/s²'
  1311 = '自動減速度Z: %d mm/s²'
  411 = '自動減速度θ:[%d]mm/s²'
  758 = '自動速度X: %d mm/s'
  665 = '自動速度Y: %d mm/s'
  1883 = '自動速度Z: %d mm/s'
  38 = '自動速度θ:[%d]mm/s'
  87 = '自動運転'
  1308 = '自動運転停止'
  987 = '自動運転開始'
  1547 = '製品データを保存します。'
  893 = '製品名'
  625 = '製品登録'
  1045 = '設定'
  945 = '設定テーブル位置:\u3000%s'
  1716 = '設定時刻'
  309 = '設定時刻に自動で'
  2028 = '設定時刻に自動でサンプルを取ります。'
  199 = '詳細'
  811 = '識別コード'
  1771 = '近接センサ値'
  132 = '通過位置'
  1078 = '速度'
  801 = '速度㎜/ｓ'
  329 = '開'
  897 = '開始キャビ'
  626 = '電磁弁'
  556 = '電磁弁操作'
  1474 = '＊24時表記'
  1138 = '＊Additional modeが有効になっていません＊'
  8 = '＊ゲート測定器原点出しを行います。'
  21 = '＊ターゲット距離からの相対距離'
  727 = '＊プログラムをリセットします'
  821 = '＊マイナス値は規格外値'
END_TEXTLIST

// ---- VISUs/Dialog/d_gm_saveBtn.TcVIS
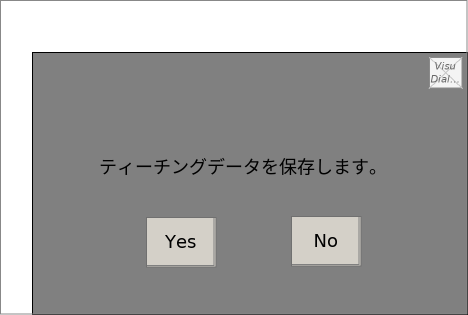
VISUALIZATION d_gm_saveBtn  // 468x315
    Rectangle (32,52 436x263)
    Image (429,57 33x31), image: VisuDialogs.ImagePoolDialogs.Delete
        OnMouseClick: CloseDialog Dialog=d_gm_saveBtn, Result=OK, NumpadKeypadSet=True
    Label (56,140 374x55), "ティーチングデータを保存します。"
    Button (146,217 70x50), "Yes"
        tap gvl_visu.flg_btn_rotaryPos
        OnMouseClick: CloseDialog Dialog=d_gm_saveBtn, Result=OK, NumpadKeypadSet=True
    Button (291,216 70x50), "No"
        OnMouseClick: CloseDialog Dialog=d_gm_saveBtn, Result=OK, NumpadKeypadSet=True
END_VISUALIZATION

// ---- VISUs/Dialog/d_palletizeReset.TcVIS
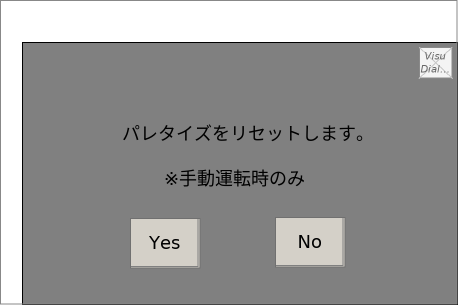
VISUALIZATION d_palletizeReset  // 458x305
    Rectangle (22,42 436x263)
    Image (419,47 33x31), image: VisuDialogs.ImagePoolDialogs.Delete
        OnMouseClick: CloseDialog Dialog=d_palletizeReset, Result=OK, NumpadKeypadSet=True
    Button (130,218 70x50), "Yes"
        tap gvl_visu.flg_btn_clrPockertQty
        OnMouseClick: CloseDialog Dialog=d_palletizeReset, Result=OK, NumpadKeypadSet=True
    Button (275,217 70x50), "No"
        OnMouseClick: CloseDialog Dialog=d_palletizeReset, Result=OK, NumpadKeypadSet=True
    Label (66,105 364x58), "パレタイズをリセットします。"
    Label (67,150 335x58), "※手動運転時のみ"
END_VISUALIZATION

// ---- VISUs/Dialog/d_preset.TcVIS
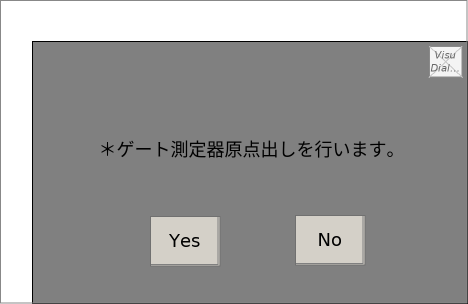
VISUALIZATION d_preset  // 468x304
    Rectangle (32,41 436x263)
    Image (429,46 33x31), image: VisuDialogs.ImagePoolDialogs.Delete
        OnMouseClick: CloseDialog Dialog=d_preset, Result=OK, NumpadKeypadSet=True
    Label (58,105 387x90), "＊ゲート測定器原点出しを行います。"
    Button (150,216 70x50), "Yes"
        tap gvl_visu.flg_btn_gateMeasurementPreset
        OnMouseClick: CloseDialog Dialog=d_preset, Result=OK, NumpadKeypadSet=True
    Button (295,215 70x50), "No"
        OnMouseClick: CloseDialog Dialog=d_preset, Result=OK, NumpadKeypadSet=True
END_VISUALIZATION

// ---- VISUs/Dialog/d_resetProject.TcVIS
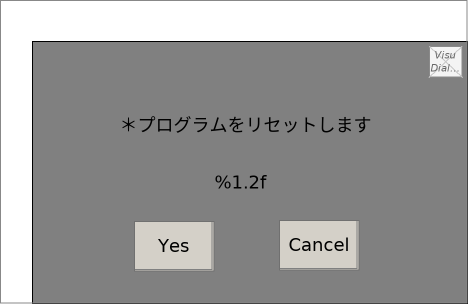
VISUALIZATION d_resetProject  // 468x304
    Rectangle (32,41 436x263)
    Image (429,46 33x31), image: VisuDialogs.ImagePoolDialogs.Delete
        OnMouseClick: CloseDialog Dialog=d_resetProject, Result=OK, NumpadKeypadSet=True
        OnMouseClick: execute { gvl_visu.flg_btn_projectReset := FALSE; }
    Label (57,93 377x65), "＊プログラムをリセットします"
    Button (134,221 80x50), "Yes", colour toggle: gvl_visu.flg_btn_projectReset
        toggle gvl_visu.flg_btn_projectReset
    Button (279,220 80x50), "Cancel"
        OnMouseClick: CloseDialog Dialog=d_resetProject, Result=OK, NumpadKeypadSet=True
        OnMouseClick: execute { gvl_visu.flg_btn_projectReset := FALSE; }
    Rectangle (53,157 370x51), "%1.2f", text variable: gvl_visu.var_projectResetLastTime
END_VISUALIZATION

// ---- VISUs/Dialog/d_sampleSchedule.TcVIS
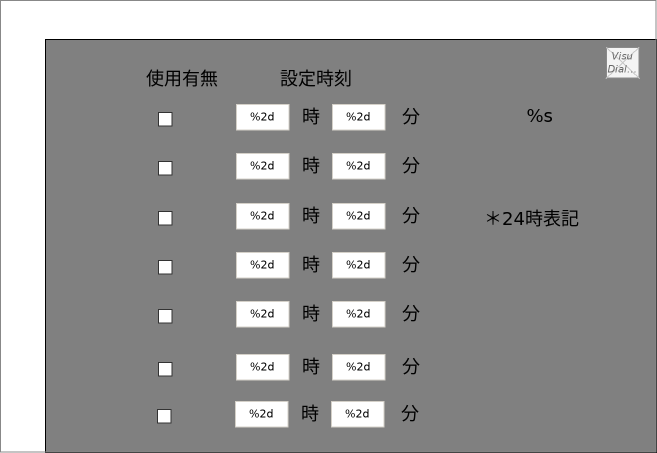
VISUALIZATION d_sampleSchedule  // 657x453
    Rectangle (45,39 612x414)
    Image (606,47 33x31), image: VisuDialogs.ImagePoolDialogs.Delete
        OnMouseClick: CloseDialog Dialog=d_sampleSchedule, Result=OK, NumpadKeypadSet=True
    Textfield (236,104 53x26), "%2d", text variable: gvl_visu.var_scheduleTimeH[0]
        OnMouseClick: write gvl_visu.var_scheduleTimeH[0] via VisuDialogs.Numpad, min 0, max 23
    Textfield (332,104 53x26), "%2d", text variable: gvl_visu.var_scheduleTimeM[0]
        OnMouseClick: write gvl_visu.var_scheduleTimeM[0] via VisuDialogs.Numpad, min 0, max 59
    Checkbox (156,104 27x30), variable: gvl_visu.var_enableSchedule[0]
    Label (291,104 40x26), "時"
    Label (391,104 40x26), "分"
    Label (253,66 126x26), "設定時刻"
    Label (119,66 126x26), "使用有無"
    Textfield (236,153 53x26), "%2d", text variable: gvl_visu.var_scheduleTimeH[1]
        OnMouseClick: write gvl_visu.var_scheduleTimeH[1] via VisuDialogs.Numpad, min 0, max 23
    Textfield (332,153 53x26), "%2d", text variable: gvl_visu.var_scheduleTimeM[1]
        OnMouseClick: write gvl_visu.var_scheduleTimeM[1] via VisuDialogs.Numpad, min 0, max 59
    Checkbox (156,153 27x30), variable: gvl_visu.var_enableSchedule[1]
    Label (291,153 40x26), "時"
    Label (391,153 40x26), "分"
    Textfield (236,203 53x26), "%2d", text variable: gvl_visu.var_scheduleTimeH[2]
        OnMouseClick: write gvl_visu.var_scheduleTimeH[2] via VisuDialogs.Numpad, min 0, max 23
    Textfield (332,203 53x26), "%2d", text variable: gvl_visu.var_scheduleTimeM[2]
        OnMouseClick: write gvl_visu.var_scheduleTimeM[2] via VisuDialogs.Numpad, min 0, max 59
    Checkbox (156,203 27x30), variable: gvl_visu.var_enableSchedule[2]
    Label (291,203 40x26), "時"
    Label (391,203 40x26), "分"
    Textfield (236,252 53x26), "%2d", text variable: gvl_visu.var_scheduleTimeH[3]
        OnMouseClick: write gvl_visu.var_scheduleTimeH[3] via VisuDialogs.Numpad, min 0, max 23
    Textfield (332,252 53x26), "%2d", text variable: gvl_visu.var_scheduleTimeM[3]
        OnMouseClick: write gvl_visu.var_scheduleTimeM[3] via VisuDialogs.Numpad, min 0, max 59
    Checkbox (156,252 27x30), variable: gvl_visu.var_enableSchedule[3]
    Label (291,252 40x26), "時"
    Label (391,252 40x26), "分"
    Textfield (236,301 53x26), "%2d", text variable: gvl_visu.var_scheduleTimeH[4]
        OnMouseClick: write gvl_visu.var_scheduleTimeH[4] via VisuDialogs.Numpad, min 0, max 23
    Textfield (332,301 53x26), "%2d", text variable: gvl_visu.var_scheduleTimeM[4]
        OnMouseClick: write gvl_visu.var_scheduleTimeM[4] via VisuDialogs.Numpad, min 0, max 59
    Checkbox (156,301 27x30), variable: gvl_visu.var_enableSchedule[4]
    Label (291,301 40x26), "時"
    Label (391,301 40x26), "分"
    Textfield (236,354 53x26), "%2d", text variable: gvl_visu.var_scheduleTimeH[5]
        OnMouseClick: write gvl_visu.var_scheduleTimeH[5] via VisuDialogs.Numpad, min 0, max 23
    Textfield (332,354 53x26), "%2d", text variable: gvl_visu.var_scheduleTimeM[5]
        OnMouseClick: write gvl_visu.var_scheduleTimeM[5] via VisuDialogs.Numpad, min 0, max 59
    Checkbox (156,354 27x30), variable: gvl_visu.var_enableSchedule[5]
    Label (291,354 40x26), "時"
    Label (391,354 40x26), "分"
    Textfield (235,401 53x26), "%2d", text variable: gvl_visu.var_scheduleTimeH[6]
        OnMouseClick: write gvl_visu.var_scheduleTimeH[6] via VisuDialogs.Numpad, min 0, max 23
    Textfield (331,401 53x26), "%2d", text variable: gvl_visu.var_scheduleTimeM[6]
        OnMouseClick: write gvl_visu.var_scheduleTimeM[6] via VisuDialogs.Numpad, min 0, max 59
    Checkbox (155,401 27x30), variable: gvl_visu.var_enableSchedule[6]
    Label (290,401 40x26), "時"
    Label (390,401 40x26), "分"
    Label (455,206 153x26), "＊24時表記"
    RoundedRectangle (426,101 228x30), "%s", text variable: gvl_visu.var_DT
END_VISUALIZATION

// ---- VISUs/Dialog/d_saveBtn.TcVIS
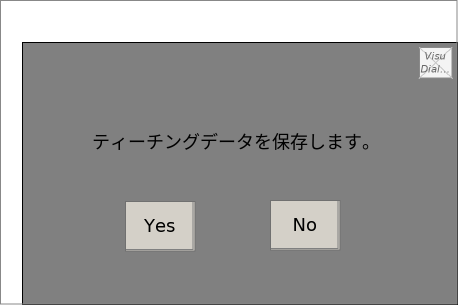
VISUALIZATION d_saveBtn  // 458x305
    Rectangle (22,42 436x263)
    Image (419,47 33x31), image: VisuDialogs.ImagePoolDialogs.Delete
        OnMouseClick: CloseDialog Dialog=d_saveBtn, Result=OK, NumpadKeypadSet=True
    Label (60,115 352x55), "ティーチングデータを保存します。"
    Button (125,201 70x50), "Yes"
        tap gvl_visu.flg_btn_savePalletize
        OnMouseClick: CloseDialog Dialog=d_saveBtn, Result=OK, NumpadKeypadSet=True
    Button (270,200 70x50), "No"
        OnMouseClick: CloseDialog Dialog=d_saveBtn, Result=OK, NumpadKeypadSet=True
END_VISUALIZATION

// ---- VISUs/Dialog/d_saveProduct.TcVIS
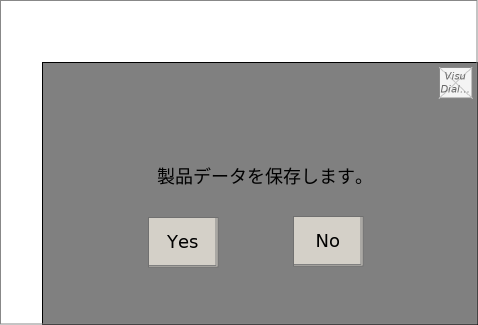
VISUALIZATION d_saveProduct  // 478x325
    Rectangle (42,62 436x263)
    Image (439,67 33x31), image: VisuDialogs.ImagePoolDialogs.Delete
        OnMouseClick: CloseDialog Dialog=d_saveProduct, Result=OK, NumpadKeypadSet=True
    Label (69,146 392x62), "製品データを保存します。"
    Button (148,217 70x50), "Yes"
        tap gvl_visu.flg_btn_saveProductInfo
        OnMouseClick: CloseDialog Dialog=d_saveProduct, Result=OK, NumpadKeypadSet=True
    Button (293,216 70x50), "No"
        OnMouseClick: CloseDialog Dialog=d_saveProduct, Result=OK, NumpadKeypadSet=True
END_VISUALIZATION

// ---- VISUs/Dialog/d_saveSample.TcVIS
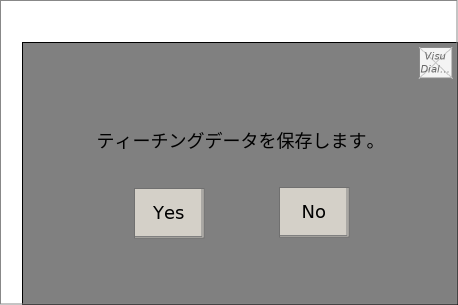
VISUALIZATION d_saveSample  // 458x305
    Rectangle (22,42 436x263)
    Image (419,47 33x31), image: VisuDialogs.ImagePoolDialogs.Delete
        OnMouseClick: CloseDialog Dialog=d_saveSample, Result=OK, NumpadKeypadSet=True
    Label (39,112 403x59), "ティーチングデータを保存します。"
    Button (134,188 70x50), "Yes"
        tap gvl_visu.flg_btn_saveSample
        OnMouseClick: CloseDialog Dialog=d_saveSample, Result=OK, NumpadKeypadSet=True
    Button (279,187 70x50), "No"
        OnMouseClick: CloseDialog Dialog=d_saveSample, Result=OK, NumpadKeypadSet=True
END_VISUALIZATION

// ---- VISUs/Dialog/d_teahingDetail.TcVIS
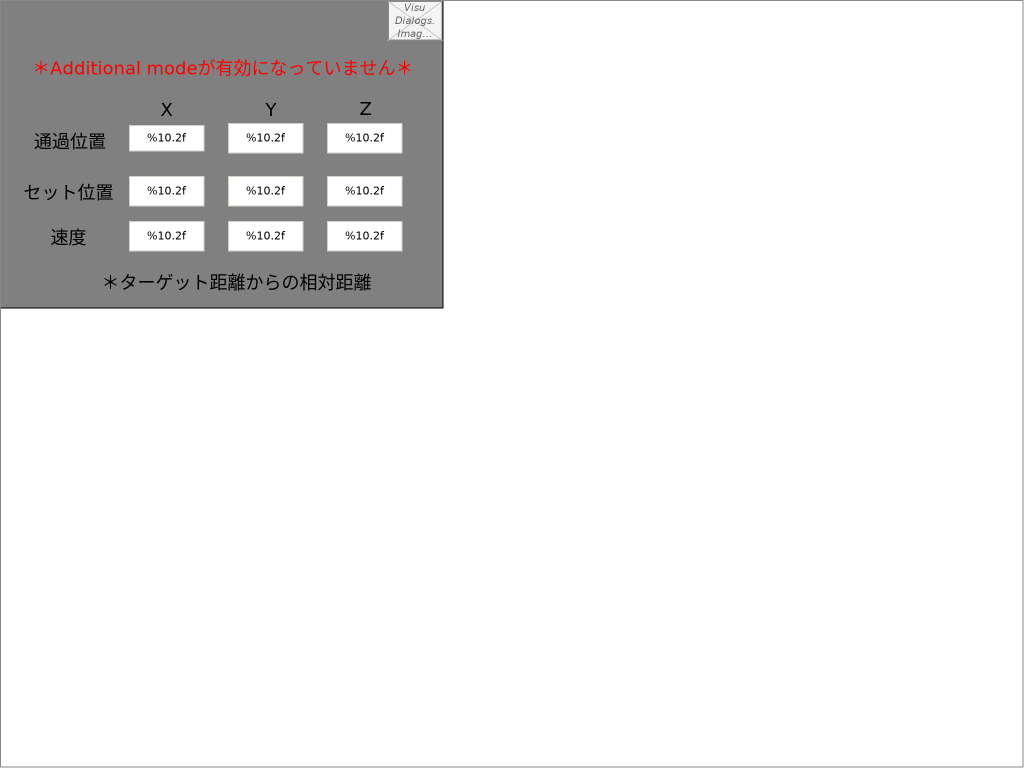
VISUALIZATION d_teahingDetail  // 1024x768
    Rectangle (0,0 443x308)
    Textfield (129,125 75x26), "%10.2f", text variable: gvl_visu.var_in_teachingDetail.passingPos.x
        OnMouseClick: write gvl_visu.var_in_teachingDetail.passingPos.x via VisuDialogs.Numpad, min -5, max 5
    Textfield (129,176 75x30), "%10.2f", text variable: gvl_visu.var_in_teachingDetail.settingPos.x
        OnMouseClick: write gvl_visu.var_in_teachingDetail.settingPos.x via VisuDialogs.Numpad, min -5, max 5
    Textfield (228,123 75x30), "%10.2f", text variable: gvl_visu.var_in_teachingDetail.passingPos.y
        OnMouseClick: write gvl_visu.var_in_teachingDetail.passingPos.y via VisuDialogs.Numpad, min -5, max 5
    Textfield (327,123 75x30), "%10.2f", text variable: gvl_visu.var_in_teachingDetail.passingPos.z
        OnMouseClick: write gvl_visu.var_in_teachingDetail.passingPos.z via VisuDialogs.Numpad, min -5, max 5
    Textfield (228,176 75x30), "%10.2f", text variable: gvl_visu.var_in_teachingDetail.settingPos.y
        OnMouseClick: write gvl_visu.var_in_teachingDetail.settingPos.y via VisuDialogs.Numpad, min -5, max 5
    Textfield (327,176 75x30), "%10.2f", text variable: gvl_visu.var_in_teachingDetail.settingPos.z
        OnMouseClick: write gvl_visu.var_in_teachingDetail.settingPos.z via VisuDialogs.Numpad, min -5, max 5
    Image (388,1 54x39), image: VisuDialogs.ImagePoolDialogs.Delete
        OnMouseClick: CloseDialog Dialog=d_teahingDetail, Result=OK, NumpadKeypadSet=True
    Label (18,178 101x30), "セット位置"
    Label (19,127 102x30), "通過位置"
    Label (125,95 84x30), "X"
    Label (324,94 84x30), "Z"
    Label (229,95 84x30), "Y"
    Label (71,260 331x46), "＊ターゲット距離からの相対距離"
    Label (16,48 414x41), "＊Additional modeが有効になっていません＊", invisible if: gvl_visu.var_dev_palletizingMode
    Textfield (129,221 75x30), "%10.2f", text variable: gvl_visu.var_in_teachingDetailVels.x.vel
        OnMouseClick: write gvl_visu.var_in_teachingDetailVels.x.vel via VisuDialogs.Numpad
    Textfield (228,221 75x30), "%10.2f", text variable: gvl_visu.var_in_teachingDetailVels.y.vel
        OnMouseClick: write gvl_visu.var_in_teachingDetailVels.y.vel via VisuDialogs.Numpad
    Textfield (327,221 75x30), "%10.2f", text variable: gvl_visu.var_in_teachingDetailVels.z.vel
        OnMouseClick: write gvl_visu.var_in_teachingDetailVels.z.vel via VisuDialogs.Numpad
    Label (18,223 101x30), "速度"
END_VISUALIZATION

// ---- VISUs/Sheet/s_debug.TcVIS
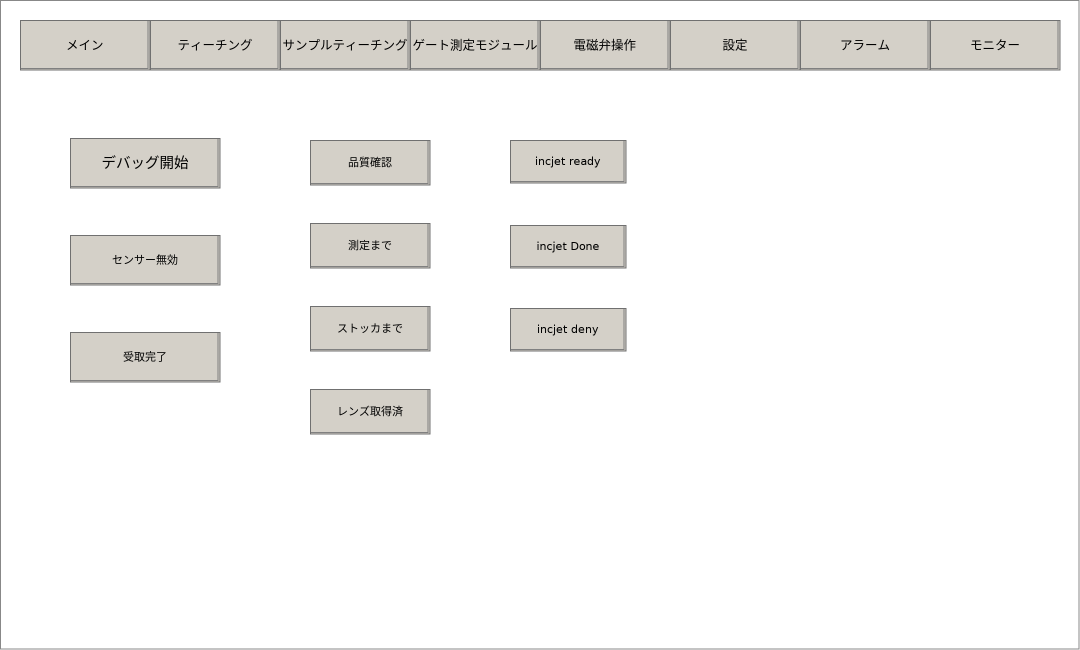
VISUALIZATION s_debug  // 1080x650
    Rectangle (0,0 1080x650)
    Button (20,20 130x50), "メイン"
        OnMouseClick: change screen: s_auto
    Button (150,20 130x50), "ティーチング"
        OnMouseClick: change screen: s_teaching1
    Button (670,20 130x50), "設定"
        OnMouseClick: change screen: s_setting
    Button (540,20 130x50), "電磁弁操作"
        OnMouseClick: change screen: s_manual
    Button (410,20 130x50), "ゲート測定モジュール"
        OnMouseClick: change screen: s_gm_teaching
    Button (800,20 130x50), "アラーム", colour toggle: gvl_io.flg_signalTowerRed
        OnMouseClick: change screen: s_alarm
    Button (280,20 130x50), "サンプルティーチング"
        OnMouseClick: change screen: s_sample
    Button (930,20 130x50), "モニター"
        OnMouseClick: change screen: s_monitor
    Button (70,235 150x50), "センサー無効", colour toggle: gvl_visu.flg_btn_vacSensOn, invisible if: NOT (gvl_debug.flg_debug_run AND gvl_param.var_currentMode = eP_programMode.auto), input disabled if: gvl_visu.flg_btn_vacSensOn
        toggle gvl_visu.flg_btn_vacSensOn
    Button (70,138 150x50), "デバッグ開始", colour toggle: gvl_debug.flg_debug_run, invisible if: NOT (gvl_param.var_currentMode = eP_programMode.auto), input disabled if: gvl_debug.flg_debug_run
        toggle gvl_debug.flg_debug_run
    Button (510,140 116x43), "incjet ready", colour toggle: gvl_debug.flg_stampReady, invisible if: NOT gvl_visu.flg_usingTimeStamp
        toggle gvl_debug.flg_stampReady
    Button (510,225 116x43), "incjet Done", colour toggle: gvl_debug.flg_stampDone, invisible if: NOT gvl_visu.flg_usingTimeStamp
        tap gvl_debug.flg_stampDone
    Button (510,308 116x43), "incjet deny", colour toggle: gvl_gm.var_incjetInfo.flg_denyStamp, invisible if: NOT gvl_visu.flg_usingTimeStamp
        toggle gvl_gm.var_incjetInfo.flg_denyStamp
    Button (310,223 120x45), "測定まで", colour toggle: gvl_debug.flg_to_measurement, invisible if: NOT (gvl_param.var_currentMode = eP_programMode.auto AND gvl_debug.flg_check_quality)
        toggle gvl_debug.flg_to_measurement
    Button (310,306 120x45), "ストッカまで", colour toggle: gvl_debug.flg_to_stocker, invisible if: NOT (gvl_param.var_currentMode = eP_programMode.auto AND gvl_debug.flg_check_quality)
        toggle gvl_debug.flg_to_stocker
    Button (310,389 120x45), "レンズ取得済", colour toggle: gvl_debug.flg_to_acquired, invisible if: NOT gvl_debug.flg_to_demand
        tap gvl_debug.flg_to_acquired
    Button (310,140 120x45), "品質確認", colour toggle: gvl_debug.flg_check_quality, invisible if: NOT (gvl_param.var_currentMode = eP_programMode.auto)
        toggle gvl_debug.flg_check_quality
    Button (70,332 150x50), "受取完了", invisible if: gvl_visu.flg_btn_vacSensOn OR NOT gvl_debug.out_busy OR NOT gvl_io.in_wire_gm_fiberSens
        tap gvl_visu.flg_btn_lensSetDone
END_VISUALIZATION

// ---- VISUs/Sheet/s_gateLengthData.TcVIS
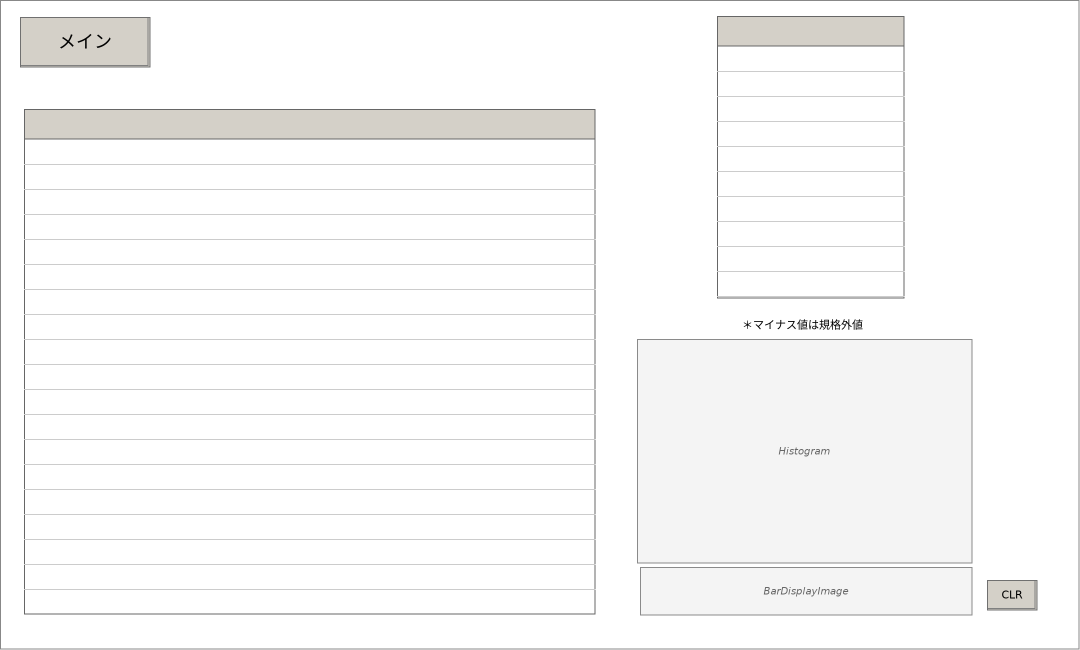
VISUALIZATION s_gateLengthData  // 1080x650
    Rectangle (0,0 1080x650)
        OnMouseClick: change screen: Previous 
    Table (717,16 187x282), data array: gvl_visu.var_gateLengthList
        p3854506369: gvl_visu.var_gateLengthList[INDEX]
        p2232123230: ゲート長さ
    Histogram (637,339 335x224), scale format: %.1f, scale -3..3
        p1518820177: gvl_visu.var_gateLengthList
        p102497268: gvl_visu.var_gateLengthList
        p788070771: ARRAY [0..49] OF REAL
    BarDisplayImage (640,567 332x48), value: gvl_visu.var_curenntGateData, style: BarDisplayImage-Gray, scale format: %.1f, scale 0..3
    Button (20,17 130x50), "メイン"
        OnMouseClick: change screen: s_auto
    Label (739,310 150x30), "＊マイナス値は規格外値"
    Table (24,109 571x505), data array: gvl_visu.var_gateLengthListCav
        p3854506369: gvl_visu.var_gateLengthListCav[1][INDEX]
        p1892666644: gvl_visu.var_gateLengthListCav[2][INDEX]
        p338671338: gvl_visu.var_gateLengthListCav[3][INDEX]
        p2170511999: gvl_visu.var_gateLengthListCav[4][INDEX]
        p3723444502: gvl_visu.var_gateLengthListCav[5][INDEX]
        p1218418051: gvl_visu.var_gateLengthListCav[6][INDEX]
        p746581629: gvl_visu.var_gateLengthListCav[7][INDEX]
        p3104783080: gvl_visu.var_gateLengthListCav[8][INDEX]
        p2232123230: Cav1
        p511219082: Cav2
        p1755163831: Cav3
        p4092479075: Cav4
        p2237128397: Cav5
        p505689113: Cav6
        p1757482276: Cav7
        p4088588272: Cav8
    Button (987,580 50x30), "CLR"
        tap gvl_visu.flg_btn_clrGateData
END_VISUALIZATION

// ---- VISUs/Sheet/s_manual.TcVIS
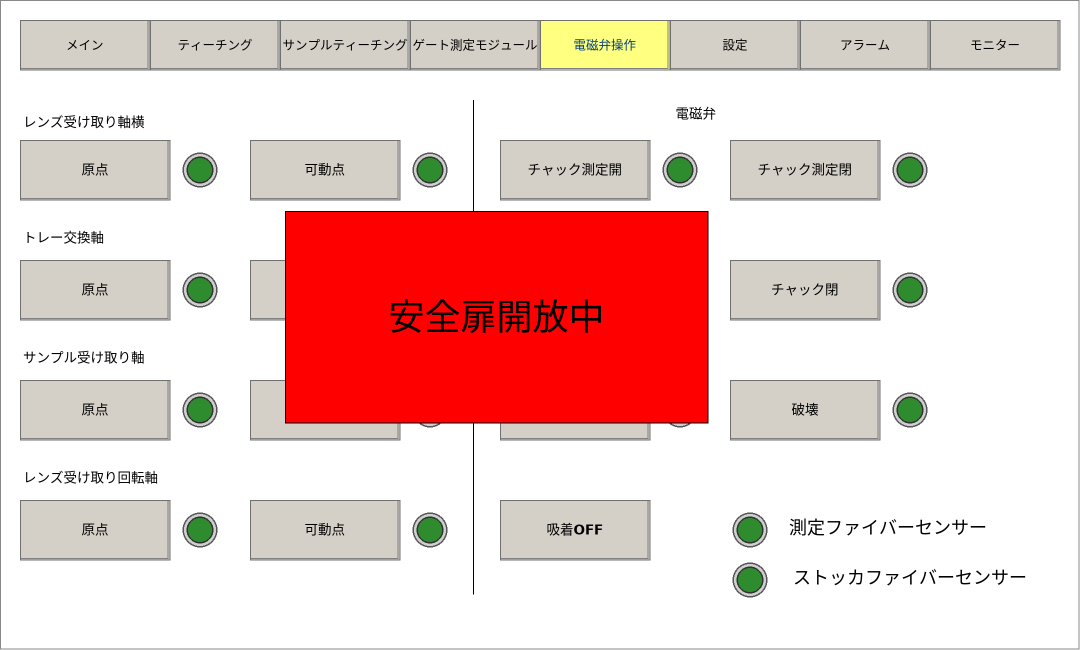
VISUALIZATION s_manual  // 1080x650
    Rectangle (0,0 1080x650)
    Button (20,140 150x60), "原点"
        tap gvl_visu.flg_btn_eleTransportNegative
    Button (20,260 150x60), "原点"
        tap gvl_visu.flg_btn_eleTrayChangeNegative
    Lamp1 (180,150 40x40), variable: gvl_elecylinder.ref_axis_transport.input.in_flg_sensA, style: Lamp-Lamp1-Green
    Lamp1 (180,270 40x40), variable: gvl_elecylinder.ref_axis_trayChange.input.in_flg_sensA, style: Lamp-Lamp1-Green
    Button (250,140 150x60), "可動点"
        tap gvl_visu.flg_btn_eleTransportPostive
    Button (250,260 150x60), "可動点"
        tap gvl_visu.flg_btn_eleTrayChangePositive
    Lamp1 (410,150 40x40), variable: gvl_elecylinder.ref_axis_transport.input.in_flg_sensB, style: Lamp-Lamp1-Green
    Lamp1 (410,270 40x40), variable: gvl_elecylinder.ref_axis_trayChange.input.in_flg_sensB, style: Lamp-Lamp1-Green
    Button (500,140 150x60), "チャック測定開"
        tap gvl_visu.flg_btn_svChuckOpen
    Button (500,260 150x60), "チャック開"
        tap gvl_visu.flg_btn_svPushOpen
    Button (730,260 150x60), "チャック閉"
        tap gvl_visu.flg_btn_svPushClose
    Lamp1 (890,150 40x40), tooltip "開", variable: gvl_solv.ref_chuck.in.in_flg_sensB, style: Lamp-Lamp1-Green
    Lamp1 (890,270 40x40), variable: gvl_solv.ref_push.in.in_flg_sensB, style: Lamp-Lamp1-Green
    Lamp1 (660,270 40x40), variable: gvl_solv.ref_push.in.in_flg_sensA, style: Lamp-Lamp1-Green
    Label (621,84 150x60), "電磁弁"
    Line (473,100) (473,594)
    Label (20,100 266x45), "レンズ受け取り軸横"
    Label (20,220 191x36), "トレー交換軸"
    Button (20,380 150x60), "原点"
        tap gvl_visu.flg_btn_eleSampleNegative
    Lamp1 (180,390 40x40), variable: gvl_elecylinder.ref_axis_sample.input.in_flg_sensA, style: Lamp-Lamp1-Green
    Button (250,380 150x60), "可動点"
        tap gvl_visu.flg_btn_eleSamplePositive
    Lamp1 (410,390 40x40), variable: gvl_elecylinder.ref_axis_sample.input.in_flg_sensB, style: Lamp-Lamp1-Green
    Label (20,340 262x36), "サンプル受け取り軸"
    Lamp1 (660,150 40x40), tooltip "開", variable: gvl_solv.ref_chuck.in.in_flg_sensA, style: Lamp-Lamp1-Green
    Label (20,460 262x36), "レンズ受け取り回転軸"
    Button (20,500 150x60), "原点"
        tap gvl_visu.flg_btn_eleRotaryNegative
    Lamp1 (180,510 40x40), variable: gvl_elecylinder.ref_axis_rotary.input.in_flg_sensA, style: Lamp-Lamp1-Green
    Button (250,500 150x60), "可動点"
        tap gvl_visu.flg_btn_eleRotaryPositive
    Lamp1 (410,510 40x40), variable: gvl_elecylinder.ref_axis_rotary.input.in_flg_sensB, style: Lamp-Lamp1-Green
    Button (730,140 150x60), "チャック測定閉"
        tap gvl_visu.flg_btn_svChuckClose
    Button (500,380 150x60), "吸着ON"
        tap gvl_visu.flg_btn_vacuumOn
    Button (730,380 150x60), "破壊"
        tap gvl_visu.flg_btn_breakOn
    Lamp1 (890,390 40x40), variable: gvl_solv.ref_ejector.input.in_flg_sensBrk, style: Lamp-Lamp1-Green
    Lamp1 (660,390 40x40), tooltip "開", variable: gvl_solv.ref_ejector.input.in_flg_sensVac, style: Lamp-Lamp1-Green
    Button (500,500 150x60), "吸着OFF"
        tap gvl_visu.flg_btn_vacuumOff
    Button (20,20 130x50), "メイン"
        OnMouseClick: change screen: s_auto
    Button (150,20 130x50), "ティーチング"
        OnMouseClick: change screen: s_teaching1
    Button (670,20 130x50), "設定"
        OnMouseClick: change screen: s_setting
    Button (540,20 130x50), "電磁弁操作"
        OnMouseClick: change screen: s_manual
    Button (410,20 130x50), "ゲート測定モジュール"
        OnMouseClick: change screen: s_gm_teaching
    Button (800,20 130x50), "アラーム", colour toggle: gvl_io.flg_signalTowerRed
        OnMouseClick: change screen: s_alarm
    Button (280,20 130x50), "サンプルティーチング"
        OnMouseClick: change screen: s_alarm
    Rectangle (285,211 423x212), "安全扉開放中", text variable: gvl_io.flg_frontSaftyDoor or gvl_param.var_currentMode <> eP_programMode.auto, invisible if: gvl_io.flg_frontSaftyDoor or gvl_param.var_currentMode <> eP_programMode.auto
    Button (930,20 130x50), "モニター"
        OnMouseClick: change screen: s_monitor
    Lamp1 (730,510 40x40), variable: gvl_io.flg_gm_fiberSens, style: Lamp-Lamp1-Green
    Lamp1 (730,560 40x40), variable: gvl_io.flg_fiberSens, style: Lamp-Lamp1-Green
    Label (786,510 235x36), "測定ファイバーセンサー"
    Label (790,560 235x36), "ストッカファイバーセンサー"
END_VISUALIZATION

// ---- VISUs/Sheet/s_addNewProduct.TcVIS
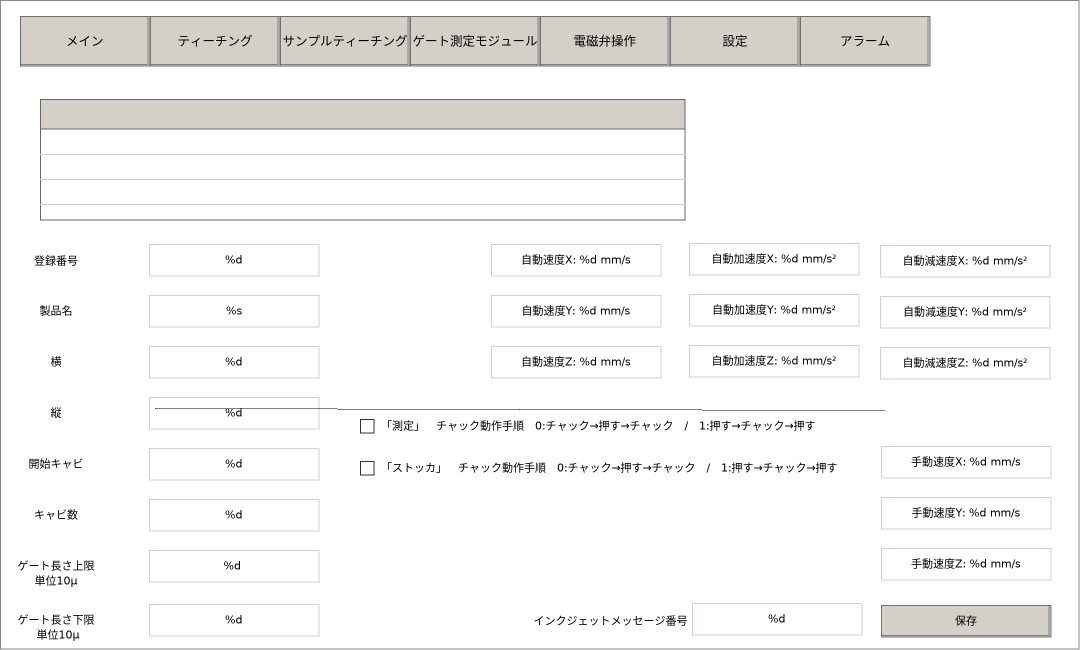
VISUALIZATION s_addNewProduct  // 1080x650
    Rectangle (0,0 1080x650)
    Textfield (149,346 170x32), "%d", text variable: gvl_visu.var_in_productGenerate.bottomPocketQty
        OnMouseClick: write gvl_visu.var_in_productGenerate.bottomPocketQty via VisuDialogs.Numpad
    Textfield (149,397 170x32), "%d", text variable: gvl_visu.var_in_productGenerate.vertivalPocketQty
        OnMouseClick: write gvl_visu.var_in_productGenerate.vertivalPocketQty via VisuDialogs.Numpad
    Textfield (149,499 170x32), "%d", text variable: gvl_visu.var_in_productGenerate.cavQty
        OnMouseClick: write gvl_visu.var_in_productGenerate.cavQty via VisuDialogs.Numpad
    Textfield (149,448 170x32), "%d", text variable: gvl_visu.var_in_productGenerate.startCav
        OnMouseClick: write gvl_visu.var_in_productGenerate.startCav via VisuDialogs.Numpad
    Label (6,398 100x30), "縦"
    Label (6,347 100x30), "横"
    Label (6,500 100x30), "キャビ数"
    Label (6,449 100x30), "開始キャビ"
    Textfield (149,295 170x32), "%s", text variable: gvl_visu.var_in_productGenerate.name
        OnMouseClick: write gvl_visu.var_in_productGenerate.name via VisuDialogs.Keypad
    Label (6,296 100x30), "製品名"
    Label (6,246 100x30), "登録番号"
    Textfield (149,244 170x32), "%d", text variable: gvl_visu.var_in_productGenerate.num
        OnMouseClick: write gvl_visu.var_in_productGenerate.num via VisuDialogs.Numpad
    Textfield (149,550 170x32), "%d", text variable: gvl_visu.var_in_productGenerate.gateLength_max
        OnMouseClick: write gvl_visu.var_in_productGenerate.gateLength_max via VisuDialogs.Numpad
    Label (6,551 100x30), "ゲート長さ上限"
    Label (6,605 100x30), "ゲート長さ下限"
    Table (40,99 645x121), data array: gvl_param.var_productInfo
        p3854506369: gvl_param.var_productInfo[INDEX].num
        p1892666644: gvl_param.var_productInfo[INDEX].name
        p338671338: gvl_param.var_productInfo[INDEX].cavQty
        p2170511999: gvl_param.var_productInfo[INDEX].bottomPocketQty
        p3723444502: gvl_param.var_productInfo[INDEX].vertivalPocketQty
        p1218418051: gvl_param.var_productInfo[INDEX].pocketSumQty
        p746581629: gvl_param.var_productInfo[INDEX].startCav
        p3104783080: gvl_param.var_productInfo[INDEX].gateLength_min
        p2501879983: gvl_param.var_productInfo[INDEX].gateLength_max
        p2232123230: 番号
        p511219082: 製品名
        p1755163831: キャビ数
        p4092479075: トレイ横数
        p2237128397: トレイ縦数
        p505689113: 入り数
        p1757482276: 開始キャビ
        p4088588272: ゲート下限
        p2243050616: ゲート上限
        p7306298: gvl_param.var_productInfo[INDEX].teachPos
        p1933151965: gvl_param.var_productInfo[INDEX].autoVels
        p3863566920: gvl_param.var_productInfo[INDEX].manaulVels
    Textfield (149,604 170x32), "%d", text variable: gvl_visu.var_in_productGenerate.gateLength_min
        OnMouseClick: write gvl_visu.var_in_productGenerate.gateLength_min via VisuDialogs.Numpad
    Textfield (491,295 170x32), "自動速度Y: %d mm/s", text variable: gvl_visu.var_in_productGenerate.autoVels.y.vel
        OnMouseClick: write gvl_visu.var_in_productGenerate.autoVels.y.vel via VisuDialogs.Numpad
    Textfield (491,346 170x32), "自動速度Z: %d mm/s", text variable: gvl_visu.var_in_productGenerate.autoVels.z.vel
        OnMouseClick: write gvl_visu.var_in_productGenerate.autoVels.z.vel via VisuDialogs.Numpad
    Textfield (881,497 170x32), "手動速度Y: %d mm/s", text variable: gvl_visu.var_in_productGenerate.manaulVels.y.vel
        OnMouseClick: write gvl_visu.var_in_productGenerate.manaulVels.y.vel via VisuDialogs.Numpad
    Textfield (881,446 170x32), "手動速度X: %d mm/s", text variable: gvl_visu.var_in_productGenerate.manaulVels.x.vel
        OnMouseClick: write gvl_visu.var_in_productGenerate.manaulVels.x.vel via VisuDialogs.Numpad
    Textfield (491,244 170x32), "自動速度X: %d mm/s", text variable: gvl_visu.var_in_productGenerate.autoVels.x.vel
        OnMouseClick: write gvl_visu.var_in_productGenerate.autoVels.x.vel via VisuDialogs.Numpad
    Textfield (881,548 170x32), "手動速度Z: %d mm/s", text variable: gvl_visu.var_in_productGenerate.manaulVels.z.vel
        OnMouseClick: write gvl_visu.var_in_productGenerate.manaulVels.z.vel via VisuDialogs.Numpad
    Button (881,605 170x32), "保存"
        tap gvl_visu.flg_btn_saveProductInfo
    Textfield (689,294 170x32), "自動加速度Y: %d mm/s²", text variable: gvl_visu.var_in_productGenerate.autoVels.y.acc
        OnMouseClick: write gvl_visu.var_in_productGenerate.autoVels.y.acc via VisuDialogs.Numpad
    Textfield (689,345 170x32), "自動加速度Z: %d mm/s²", text variable: gvl_visu.var_in_productGenerate.autoVels.z.acc
        OnMouseClick: write gvl_visu.var_in_productGenerate.autoVels.z.acc via VisuDialogs.Numpad
    Textfield (689,243 170x32), "自動加速度X: %d mm/s²", text variable: gvl_visu.var_in_productGenerate.autoVels.x.acc
        OnMouseClick: write gvl_visu.var_in_productGenerate.autoVels.x.acc via VisuDialogs.Numpad
    Textfield (880,296 170x32), "自動減速度Y: %d mm/s²", text variable: gvl_visu.var_in_productGenerate.autoVels.y.dcc
        OnMouseClick: write gvl_visu.var_in_productGenerate.autoVels.y.dcc via VisuDialogs.Numpad
    Textfield (880,347 170x32), "自動減速度Z: %d mm/s²", text variable: gvl_visu.var_in_productGenerate.autoVels.z.dcc
        OnMouseClick: write gvl_visu.var_in_productGenerate.autoVels.z.dcc via VisuDialogs.Numpad
    Textfield (880,245 170x32), "自動減速度X: %d mm/s²", text variable: gvl_visu.var_in_productGenerate.autoVels.x.dcc
        OnMouseClick: write gvl_visu.var_in_productGenerate.autoVels.x.dcc via VisuDialogs.Numpad
    Line (155,408) (884,410)
    Label (6,566 100x30), "単位10μ"
    Label (8,620 100x30), "単位10μ"
    Textfield (692,603 170x32), "%d", text variable: gvl_visu.var_in_productGenerate.incjetMsgNo
        OnMouseClick: write gvl_visu.var_in_productGenerate.incjetMsgNo via VisuDialogs.Numpad
    Label (537,606 147x30), "インクジェットメッセージ番号"
    Button (20,16 130x50), "メイン"
        OnMouseClick: change screen: s_auto
    Button (150,16 130x50), "ティーチング"
        OnMouseClick: change screen: s_teaching1
    Button (670,16 130x50), "設定"
        OnMouseClick: change screen: s_setting
    Button (540,16 130x50), "電磁弁操作"
        OnMouseClick: change screen: s_manual
    Button (410,16 130x50), "ゲート測定モジュール"
        OnMouseClick: change screen: s_gm_teaching
    Button (800,16 130x50), "アラーム", colour toggle: gvl_io.flg_signalTowerRed
        OnMouseClick: change screen: s_alarm
    Button (280,16 130x50), "サンプルティーチング"
        OnMouseClick: change screen: s_sample
    Checkbox (358,411 505x30), "「測定」 チャック動作手順 0:チャック→押す→チャック / 1:押す→チャック→押す", variable: gvl_visu.var_in_productGenerate.flg_mode_measurement
    Checkbox (358,453 503x30), "「ストッカ」 チャック動作手順 0:チャック→押す→チャック / 1:押す→チャック→押す", variable: gvl_visu.var_in_productGenerate.flg_mode_stocker
END_VISUALIZATION

// ---- VISUs/Sheet/s_alarm.TcVIS
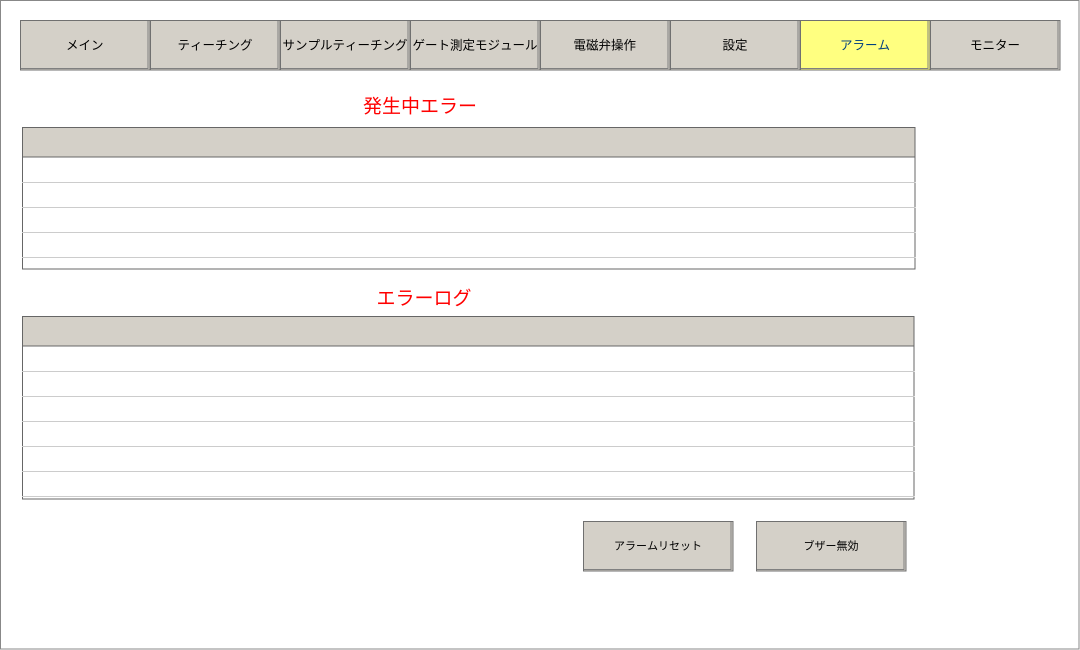
VISUALIZATION s_alarm  // 1080x650
    Rectangle (0,0 1080x650)
    Table (22,316 892x183), data array: gvl_error.var_ary_alarmlistLog
        p3854506369: gvl_error.var_ary_alarmlistLog[INDEX].var_alarmLevel
        p1892666644: gvl_error.var_ary_alarmlistLog[INDEX].var_alarmName
        p511219082: アラーム名
        p338671338: gvl_error.var_ary_alarmlistLog[INDEX].var_alarmMassge
        p2170511999: gvl_error.var_ary_alarmlistLog[INDEX].var_alarmTime
        p3723444502: gvl_error.var_ary_alarmlistLog[INDEX].var_alarmCode1
        p1218418051: gvl_error.var_ary_alarmlistLog[INDEX].var_alarmCode2
        p1755163831: 詳細
        p4092479075: 発生時刻
        p2237128397: 識別コード
        p505689113: エラーID
    Table (22,127 893x142), data array: gvl_error.var_ary_alarmlistActive
        p3854506369: gvl_error.var_ary_alarmlistActive[INDEX].var_alarmLevel
        p1892666644: gvl_error.var_ary_alarmlistActive[INDEX].var_alarmName
        p338671338: gvl_error.var_ary_alarmlistActive[INDEX].var_alarmMassge
        p2170511999: gvl_error.var_ary_alarmlistActive[INDEX].var_alarmTime
        p3723444502: gvl_error.var_ary_alarmlistActive[INDEX].var_alarmCode1
        p1218418051: gvl_error.var_ary_alarmlistActive[INDEX].var_alarmCode2
        p511219082: アラーム名
        p1755163831: 詳細
        p4092479075: 発生時刻
        p2237128397: 識別コード
        p505689113: エラーID
    Button (583,521 150x50), "アラームリセット"
        tap gvl_error.flg_reset
    Label (299,283 250x30), "エラーログ"
    Label (295,91 250x30), "発生中エラー"
    Button (20,20 130x50), "メイン"
        OnMouseClick: change screen: s_auto
    Button (150,20 130x50), "ティーチング"
        OnMouseClick: change screen: s_teaching1
    Button (670,20 130x50), "設定"
        OnMouseClick: change screen: s_setting
    Button (540,20 130x50), "電磁弁操作"
        OnMouseClick: change screen: s_manual
    Button (410,20 130x50), "ゲート測定モジュール"
        OnMouseClick: change screen: s_gm_teaching
    Button (800,20 130x50), "アラーム", colour toggle: gvl_io.flg_signalTowerRed
        OnMouseClick: change screen: s_alarm
    Button (280,20 130x50), "サンプルティーチング"
        OnMouseClick: change screen: s_sample
    Button (756,521 150x50), "ブザー無効", colour toggle: gvl_visu.flg_btn_invalidBuzzer
        toggle gvl_visu.flg_btn_invalidBuzzer
    Button (930,20 130x50), "モニター"
        OnMouseClick: change screen: s_monitor
END_VISUALIZATION

// ---- VISUs/Sheet/s_auto.TcVIS
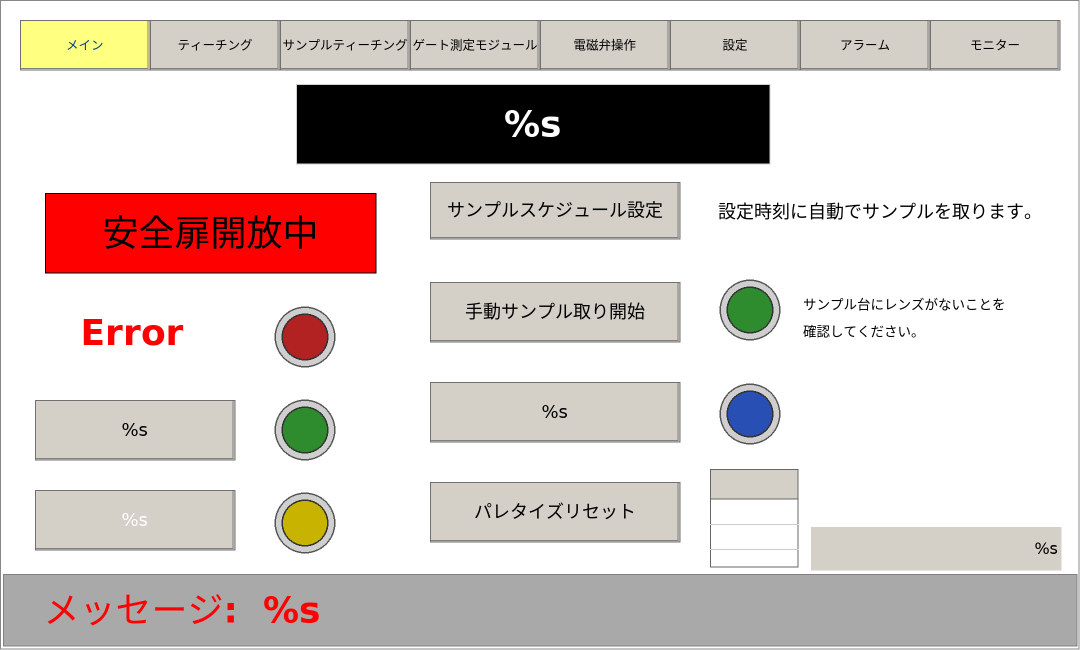
VISUALIZATION s_auto  // 1080x650
    Rectangle (0,0 1080x650)
    Button (35,400 200x60), "%s", text variable: gvl_text.var_auto_runing, colour toggle: gvl_debug.flg_debug_run AND gvl_param.var_currentMode = eP_programMode.auto
        tap gvl_visu.flg_btn_autoModeStart
    Button (35,490 200x60), "%s", text variable: gvl_text.var_stopping, colour toggle: gvl_auto.autoModeStop
        tap gvl_visu.flg_btn_autoModeStop
    Button (430,382 250x60), "%s", text variable: gvl_text.var_trayChangeDone
        toggle gvl_visu.flg_btn_trayChangeDone
    Lamp1 (715,275 70x70), variable: gvl_visu.flg_btn_sample, style: Lamp-Lamp1-Green
    Lamp1 (270,395 70x70), variable: gvl_param.var_currentMode = eP_programMode.auto, style: Lamp-Lamp1-Green
    Lamp1 (270,488 70x70), variable: gvl_param.var_currentMode = eP_programMode.manual, style: Lamp-Lamp1-Yellow
    Lamp1 (270,302 70x70), variable: gvl_param.var_currentMode = eP_programMode.error, invisible if: gvl_param.var_currentMode <> eP_programMode.error, style: Lamp-Lamp1-Red
    Label (42,293 180x79), "Error", invisible if: gvl_param.var_currentMode <> eP_programMode.error
    Lamp1 (715,379 70x70), variable: gvl_visu.flg_btn_trayChangeDone, style: Lamp-Lamp1-Blue
    RoundedRectangle (811,527 250x43), "%s", text variable: gvl_visu.var_DT
    Button (430,282 250x60), "手動サンプル取り開始"
        toggle gvl_visu.flg_btn_sample
    Rectangle (296,84 474x80), "%s", text variable: gvl_param.var_productInfo[gvl_param.var_currentProductID].name
    Rectangle (3,574 1074x72), "メッセージ: %s", text variable: gvl_visu.var_msg
    Button (430,482 250x60), "パレタイズリセット"
        OnMouseClick: OpenDialog Dialog=d_palletizeReset, OpenModal=True, OpenCentered=True
    Table (710,469 88x98), data array: gvl_auto.pocketNo
        p3854506369: gvl_auto.pocketNo[INDEX]
    Button (20,20 130x50), "メイン"
        OnMouseClick: change screen: s_auto
    Button (150,20 130x50), "ティーチング"
        OnMouseClick: change screen: s_teaching1
    Button (670,20 130x50), "設定"
        OnMouseClick: change screen: s_setting
    Button (540,20 130x50), "電磁弁操作"
        OnMouseClick: change screen: s_manual
    Button (410,20 130x50), "ゲート測定モジュール"
        OnMouseClick: change screen: s_gm_teaching
    Button (800,20 130x50), "アラーム", colour toggle: gvl_io.flg_signalTowerRed
        OnMouseClick: change screen: s_alarm
    Button (280,20 130x50), "サンプルティーチング"
        OnMouseClick: change screen: s_sample
    Button (430,182 250x57), "サンプルスケジュール設定"
        OnMouseClick: OpenDialog Dialog=d_sampleSchedule, OpenModal=True, OpenCentered=True
    Label (715,185 363x54), "設定時刻に自動でサンプルを取ります。"
    Button (930,20 130x50), "モニター"
        OnMouseClick: change screen: s_monitor
    Label (800,280 250x50), "サンプル台にレンズがないことを"
    Rectangle (45,193 331x80), "安全扉開放中", text variable: gvl_io.flg_frontSaftyDoor or gvl_param.var_currentMode <> eP_programMode.auto, invisible if: gvl_io.flg_frontSaftyDoor or gvl_param.var_currentMode <> eP_programMode.auto
    Label (800,307 250x50), "確認してください。"
END_VISUALIZATION

// ---- VISUs/Sheet/s_gm_teaching.TcVIS
